(* Schneider Machine Expert - Basic project es5_6pompe_5max_6soglie_misura_livello_scelta_alternanza_spegnimento_graduale_o_livello_minimo, file version 3.0.0.0 *)
(* ProjectInformations: Name=New project *)

HARDWARE
  Cpu 0: TM221C40R
  ModuleExtensionObject 0: TM3AI8/G
  EthernetConfiguration: NetworkName=M221, IpAllocationMode=FixedAddress, IpAddress=0.0.0.0, SubnetMask=0.0.0.0
  SerialLineConfiguration: Baud=Baud19200, Parity=ParityEven, DataBits=DataBits8, StopBits=StopBits1, PhysicalMedium=PhysicalMediumRs485, TransmissionMode=TransmissionModeModbusRtu, SlaveId=1, Addressing=SlaveAddressing
  MastTask: UsePeriodScanMode=false, PeriodScan=100
  FastTask: Period=255
  CpuBehavior: StartingMode=StartAsPreviousState, AutoSaveRamOnEeprom=true, WatchdogPeriod=250

SYMBOLS  (address, symbol, comment, settings)
  %M0       P1_USABILE
  %M1       P2_USABILE
  %M2       P1_COMANDATA  "Stesso valore di P1_CMD. Permette di identificare gli edges, visto che P1_CMD non può farlo."
  %M3       P2_COMANDATA  "Stesso valore di P2_CMD. Permette di identificare gli edges, visto che P2_CMD non può farlo."
  %M4       P3_USABILE
  %M5       P4_USABILE
  %M6       P3_COMANDATA
  %M7       P4_COMANDATA
  %M8       ESISTE_PROX_POMPA_CON_MINOR_ORE  "Nel loop, può non esistere una prossima pompa usabile e non comandata con il minor numero ore."
  %M9       ORA_E_00  "E' mezzanotte?"
  %M10      DECISO_ORDINE  "In intervallo in cui alternare le pompe per altern. giorn., è stata deciso quale sarà prossima pompa con minor ore?"
  %M11      PRIMA_POMPA_COMANDATA  "La prima pompa dell'ordine è stata effettivamente comandata quando serviva?"
  %M12      SECONDA_POMPA_COMANDATA  "La seconda pompa dell'ordine è stata effettivamente comandata quando serviva?"
  %M13      TERZA_POMPA_COMANDATA  "La terza pompa dell'ordine è stata effettivamente comandata quando serviva?"
  %M14      SOTTO_SOGLIA_MIN1
  %M15      SOPRA_SOGLIA_MAX1
  %M16      SOPRA_SOGLIA_MAX2
  %M17      PASSATO_SOGLIA_MAX1
  %M18      PASSATO_SOGLIA_MAX2
  %M19      SOTTO_SOGLIA_MIN2
  %M20      PASSATO_SOGLIA_MAX3
  %M21      PASSATO_SOGLIA_MIN3
  %M22      SOTTO_SOGLIA_MIN3
  %M23      SOPRA_SOGLIA_MAX3
  %M24      P5_USABILE
  %M25        "(occupato, placeholder)"
  %M26      P6_USABILE
  %M27      P5_COMANDATA
  %M28      P6_COMANDATA
  %M29      QUARTA_POMPA_COMANDATA
  %M30      QUINTA_POMPA_COMANDATA
  %S6       SB_TB1S  "Time base of 1 s generated by an internal clock"
  %MW0      NUM_POMPE_DA_COMANDARE  "Numero di pompe da comandare in base alle soglie raggiunte."
  %MW1      NUM_POMPE_COMANDATE  "Numero di pompe effettivamente comandate, in base alle loro disponibilità."
  %MW2      NUM_POMPE  "Numero di pompe totali."
  %MW3      ULTIMO_MINOR_SECONDI_LAVORATI  "Ultimi secondi lavorati più piccoli (valore temporaneo, da usare solo nel loop)."
  %MW4      PROSSIMA_POMPA_DA_COMANDARE  "Numero da 1 a NUM_POMPE che indica la prossima pompa da comandare."
  %MW5      POMPA_ATTUALE_LOOP  "Pompa attuale nel loop."
  %MW6      NUM_POMPE_COMANDATE_MAX  "Num"
  %MW7      CONTA_POMPE_COMANDATE_MAX  "Da usare in loop e da resettare.  Assume il valore da 1 fino a NUM_POMPE_COMANDATE_MAX."
  %MW8      ORDINE_PRIMA_POMPA
  %MW9      ORDINE_SECONDA_POMPA
  %MW10     ORDINE_TERZA_POMPA
  %MW11     STRG_ALTERNANZA_ATTUALE
  %MW12     LVL_PERC
  %MW13     ORDINE_QUARTA_POMPA
  %MW14     ORDINE_QUINTA_POMPA
  %C0       CONTATORE_P1_SECONDI_LAVORATI  [Preset=0]
  %C1       CONTATORE_P2_SECONDI_LAVORATI  [Preset=0]
  %C2       CONTATORE_P3_SECONDI_LAVORATI  [Preset=0]
  %C3       CONTATORE_P4_SECONDI_LAVORATI  [Preset=0]
  %C4       CONTATORE_P5_SECONDI_LAVORATI  [Preset=0]
  %C5       CONTATORE_P6_SECONDI_LAVORATI  [Preset=0]
  %I0.0     P1_AUTO
  %I0.1     P1_MOTO
  %I0.2     P1_ANOMALIA
  %I0.3     P2_AUTO
  %I0.4     P2_MOTO
  %I0.5     P2_ANOMALIA
  %I0.9     P3_AUTO
  %I0.10    P3_MOTO
  %I0.11    P3_ANOMALIA
  %I0.12    P4_AUTO
  %I0.13    P4_MOTO
  %I0.14    P4_ANOMALIA
  %I0.15    P5_AUTO
  %I0.16    P5_MOTO
  %I0.17    P5_ANOMALIA
  %I0.18    P6_AUTO
  %I0.19    P6_MOTO
  %I0.20    P6_ANOMALIA
  %Q0.0     P1_CMD
  %Q0.1     P2_CMD
  %Q0.2     P3_CMD
  %Q0.3     P4_CMD
  %Q0.4     ERR_STRG_ALTERNANZA_INVALIDA
  %Q0.5     P5_CMD
  %Q0.6     P6_CMD
  %IW0.0    IO_STRG_ALTERNANZA  "0 = livello minimo; 1 = spegnimento graduale;"  [Type=Type_0_10V, Scope=Scope_Normal, Minimum=0, Maximum=1000]
  %IW1.0    IO_LVL  [Type=Type_4_20mA, Scope=Scope_Customized, Minimum=4000, Maximum=20000]
  %IW1.1    SOGLIA_MIN1_PERC  [Type=Type_0_10V, Scope=Scope_Customized, Minimum=0, Maximum=100]
  %IW1.2    SOGLIA_MAX1_PERC  [Type=Type_0_10V, Scope=Scope_Customized, Minimum=0, Maximum=100]
  %IW1.3    SOGLIA_MIN2_PERC  [Type=Type_0_10V, Scope=Scope_Customized, Minimum=0, Maximum=100]
  %IW1.4    SOGLIA_MAX2_PERC  [Type=Type_0_10V, Scope=Scope_Customized, Minimum=0, Maximum=100]
  %IW1.5    SOGLIA_MIN3_PERC  [Type=Type_0_10V, Scope=Scope_Customized, Minimum=0, Maximum=100]
  %IW1.6    SOGLIA_MAX3_PERC  [Type=Type_0_10V, Scope=Scope_Customized, Minimum=0, Maximum=100]

POU Main
  (* SectionNumber=1 *)

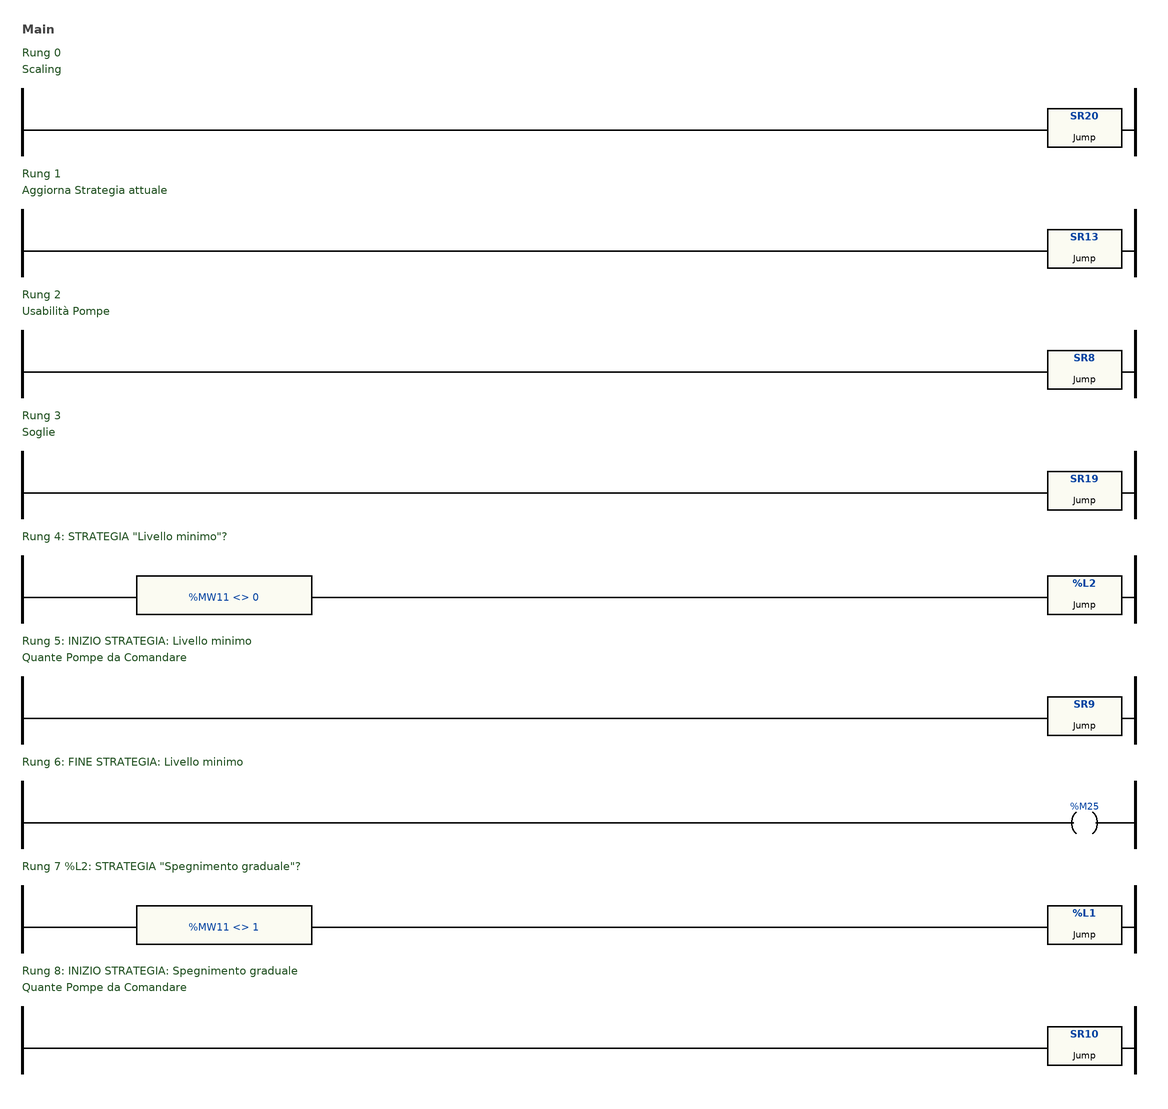

// Rung 0
// Scaling
  LD 1
  SR20
  // as ST:
  //   SR20();

// Rung 1
// Aggiorna Strategia attuale
  LD 1
  SR13
  // as ST:
  //   SR13();

// Rung 2
// Usabilità Pompe
  LD 1
  SR8
  // as ST:
  //   SR8();

// Rung 3
// Soglie
  LD 1
  SR19
  // as ST:
  //   SR19();

// Rung 4: STRATEGIA "Livello minimo"?
  LD [ %MW11 <> 0 ]       (* STRG_ALTERNANZA_ATTUALE *)
  JMPC %L2
  // as ST:
  //   IF STRG_ALTERNANZA_ATTUALE <> 0 THEN JMP %L2; END_IF;

// Rung 5: INIZIO STRATEGIA: Livello minimo
// Quante Pompe da Comandare
  LD 1
  SR9
  // as ST:
  //   SR9();

// Rung 6: FINE STRATEGIA: Livello minimo
  LD 1
  ST %M25
  // as ST:
  //   %M25 := TRUE;

// Rung 7 %L2: STRATEGIA "Spegnimento graduale"?
  %L2:
  LD [ %MW11 <> 1 ]       (* STRG_ALTERNANZA_ATTUALE *)
  JMPC %L1
  // as ST:
  //   %L2:
  //   IF STRG_ALTERNANZA_ATTUALE <> 1 THEN JMP %L1; END_IF;

// Rung 8: INIZIO STRATEGIA: Spegnimento graduale
// Quante Pompe da Comandare
  LD 1
  SR10
  // as ST:
  //   SR10();

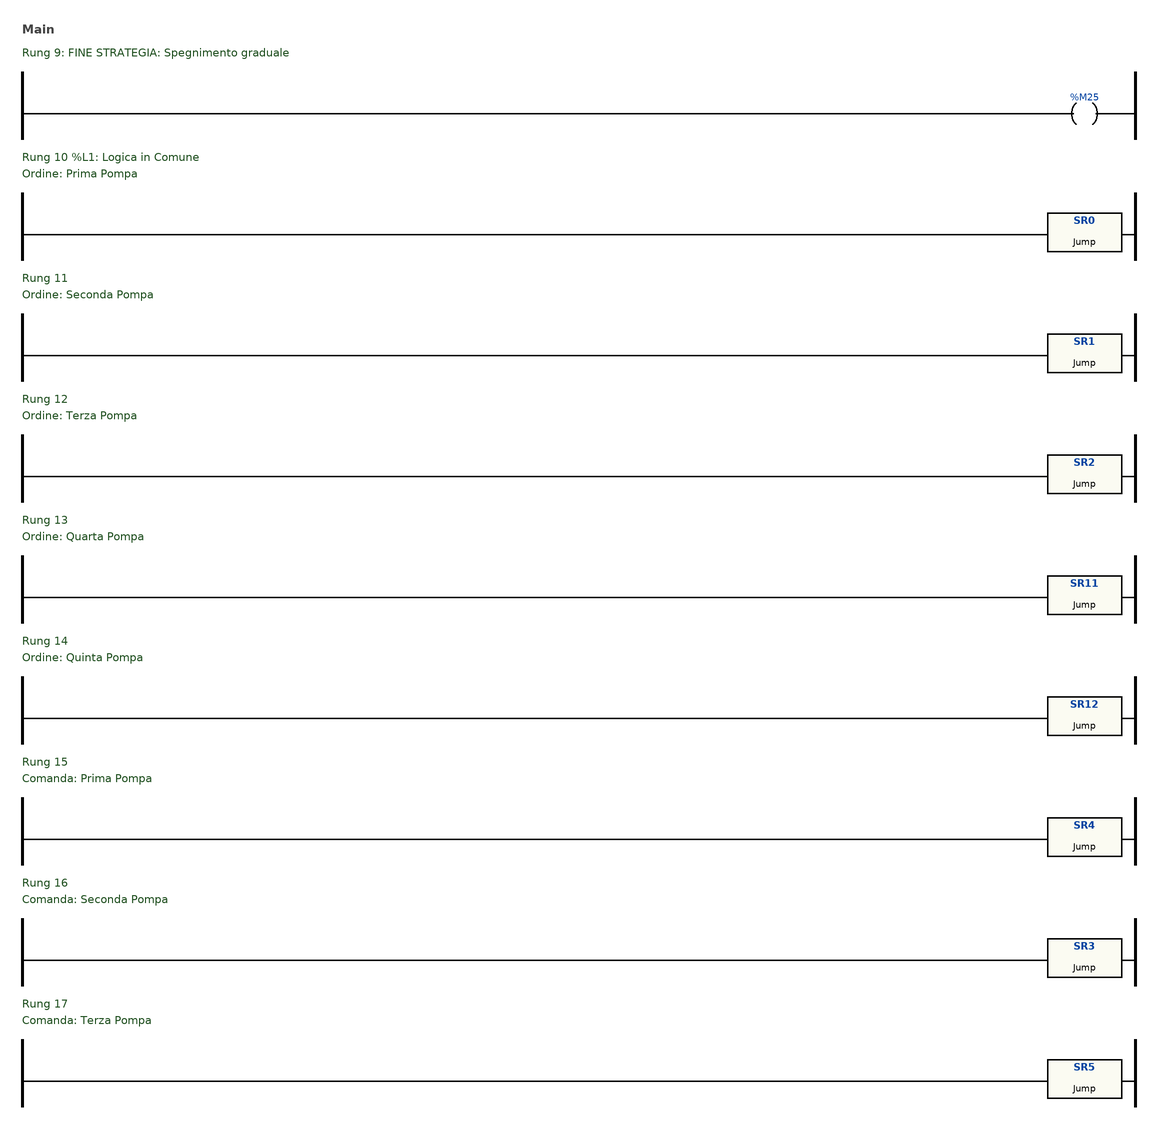

// Rung 9: FINE STRATEGIA: Spegnimento graduale
  LD 1
  ST %M25
  // as ST:
  //   %M25 := TRUE;

// Rung 10 %L1: Logica in Comune
// Ordine: Prima Pompa
  %L1:
  LD 1
  SR0
  // as ST:
  //   %L1:
  //   SR0();

// Rung 11
// Ordine: Seconda Pompa
  LD 1
  SR1
  // as ST:
  //   SR1();

// Rung 12
// Ordine: Terza Pompa
  LD 1
  SR2
  // as ST:
  //   SR2();

// Rung 13
// Ordine: Quarta Pompa
  LD 1
  SR11
  // as ST:
  //   SR11();

// Rung 14
// Ordine: Quinta Pompa
  LD 1
  SR12
  // as ST:
  //   SR12();

// Rung 15
// Comanda: Prima Pompa
  LD 1
  SR4
  // as ST:
  //   SR4();

// Rung 16
// Comanda: Seconda Pompa
  LD 1
  SR3
  // as ST:
  //   SR3();

// Rung 17
// Comanda: Terza Pompa
  LD 1
  SR5
  // as ST:
  //   SR5();

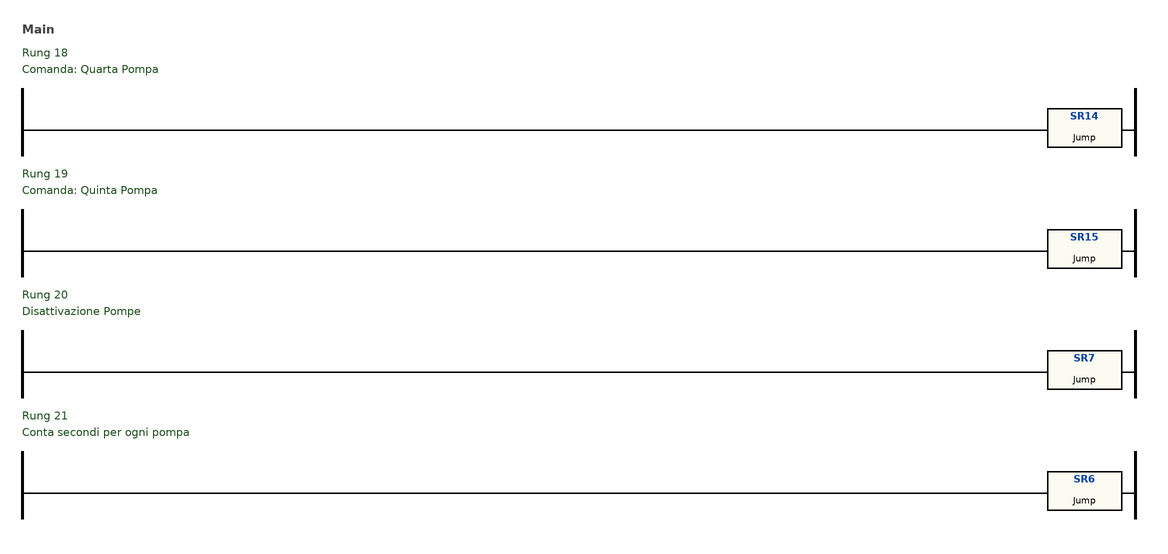

// Rung 18
// Comanda: Quarta Pompa
  LD 1
  SR14
  // as ST:
  //   SR14();

// Rung 19
// Comanda: Quinta Pompa
  LD 1
  SR15
  // as ST:
  //   SR15();

// Rung 20
// Disattivazione Pompe
  LD 1
  SR7
  // as ST:
  //   SR7();

// Rung 21
// Conta secondi per ogni pompa
  LD 1
  SR6
  // as ST:
  //   SR6();

Subroutine Ordine: Prima Pompa
  (* SectionNumber=2, Number=0 *)

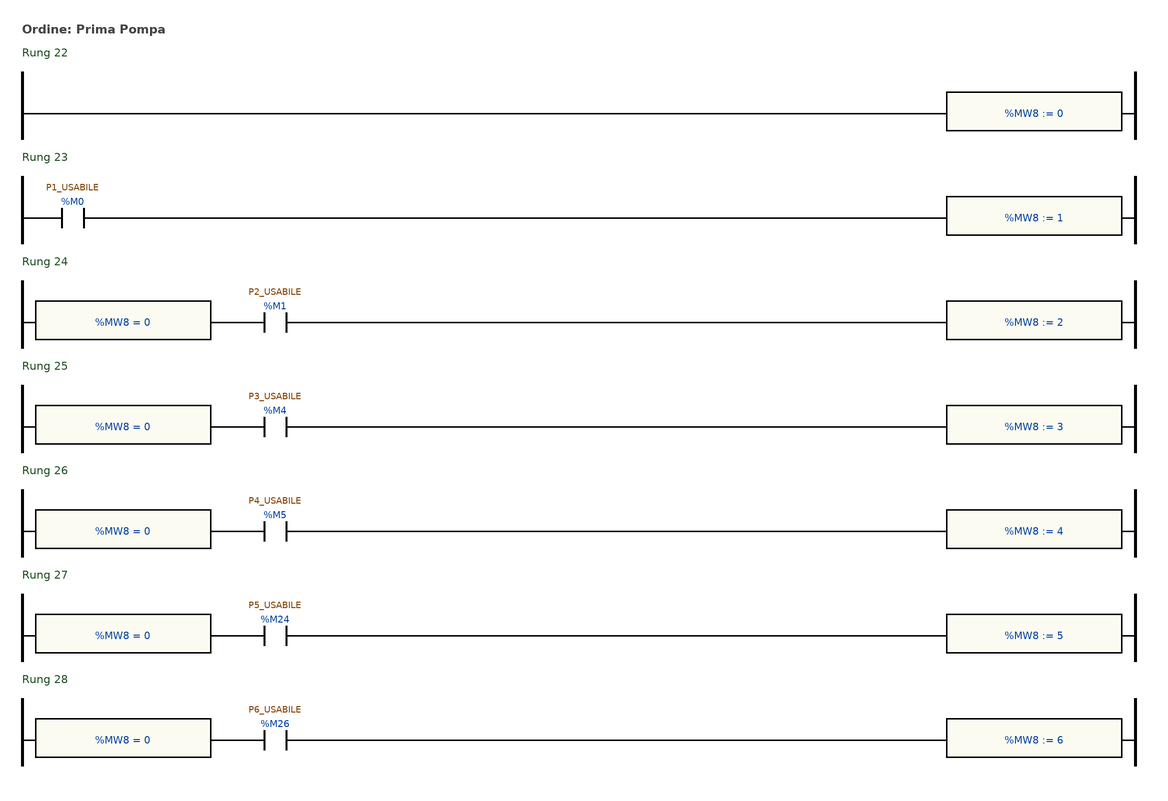

// Rung 22
  LD 1
  [ %MW8 := 0 ]           (* ORDINE_PRIMA_POMPA *)
  // as ST:
  //   ORDINE_PRIMA_POMPA := 0;

// Rung 23
  LD %M0                  (* P1_USABILE *)
  [ %MW8 := 1 ]           (* ORDINE_PRIMA_POMPA *)
  // as ST:
  //   IF P1_USABILE THEN ORDINE_PRIMA_POMPA := 1; END_IF;

// Rung 24
  LD [ %MW8 = 0 ]         (* ORDINE_PRIMA_POMPA *)
  AND %M1                 (* P2_USABILE *)
  [ %MW8 := 2 ]           (* ORDINE_PRIMA_POMPA *)
  // as ST:
  //   IF ORDINE_PRIMA_POMPA = 0 AND P2_USABILE THEN ORDINE_PRIMA_POMPA := 2; END_IF;

// Rung 25
  LD [ %MW8 = 0 ]         (* ORDINE_PRIMA_POMPA *)
  AND %M4                 (* P3_USABILE *)
  [ %MW8 := 3 ]           (* ORDINE_PRIMA_POMPA *)
  // as ST:
  //   IF ORDINE_PRIMA_POMPA = 0 AND P3_USABILE THEN ORDINE_PRIMA_POMPA := 3; END_IF;

// Rung 26
  LD [ %MW8 = 0 ]         (* ORDINE_PRIMA_POMPA *)
  AND %M5                 (* P4_USABILE *)
  [ %MW8 := 4 ]           (* ORDINE_PRIMA_POMPA *)
  // as ST:
  //   IF ORDINE_PRIMA_POMPA = 0 AND P4_USABILE THEN ORDINE_PRIMA_POMPA := 4; END_IF;

// Rung 27
  LD [ %MW8 = 0 ]         (* ORDINE_PRIMA_POMPA *)
  AND %M24                (* P5_USABILE *)
  [ %MW8 := 5 ]           (* ORDINE_PRIMA_POMPA *)
  // as ST:
  //   IF ORDINE_PRIMA_POMPA = 0 AND P5_USABILE THEN ORDINE_PRIMA_POMPA := 5; END_IF;

// Rung 28
  LD [ %MW8 = 0 ]         (* ORDINE_PRIMA_POMPA *)
  AND %M26                (* P6_USABILE *)
  [ %MW8 := 6 ]           (* ORDINE_PRIMA_POMPA *)
  // as ST:
  //   IF ORDINE_PRIMA_POMPA = 0 AND P6_USABILE THEN ORDINE_PRIMA_POMPA := 6; END_IF;

Subroutine Ordine: Seconda Pompa
  (* SectionNumber=3, Number=1 *)

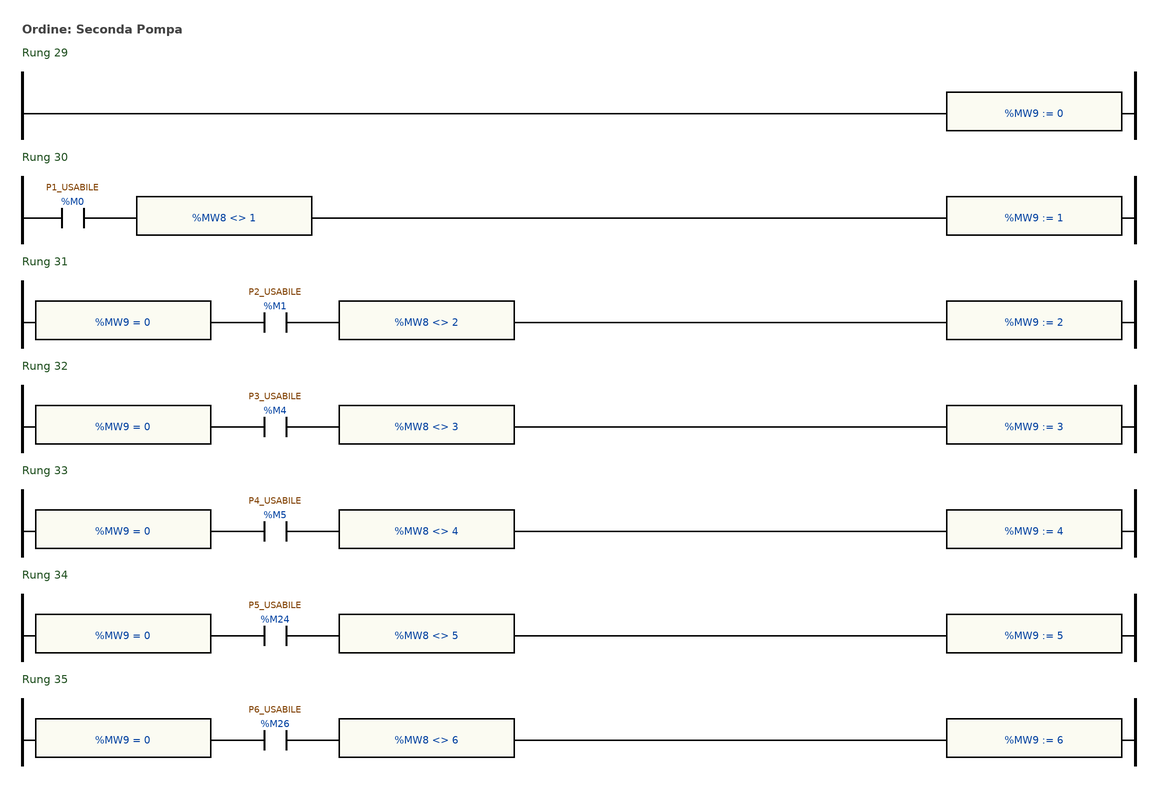

// Rung 29
  LD 1
  [ %MW9 := 0 ]           (* ORDINE_SECONDA_POMPA *)
  // as ST:
  //   ORDINE_SECONDA_POMPA := 0;

// Rung 30
  LD %M0                  (* P1_USABILE *)
  AND [ %MW8 <> 1 ]       (* ORDINE_PRIMA_POMPA *)
  [ %MW9 := 1 ]           (* ORDINE_SECONDA_POMPA *)
  // as ST:
  //   IF P1_USABILE AND ORDINE_PRIMA_POMPA <> 1 THEN ORDINE_SECONDA_POMPA := 1; END_IF;

// Rung 31
  LD [ %MW9 = 0 ]         (* ORDINE_SECONDA_POMPA *)
  AND %M1                 (* P2_USABILE *)
  AND [ %MW8 <> 2 ]       (* ORDINE_PRIMA_POMPA *)
  [ %MW9 := 2 ]           (* ORDINE_SECONDA_POMPA *)
  // as ST:
  //   IF ORDINE_SECONDA_POMPA = 0 AND P2_USABILE AND ORDINE_PRIMA_POMPA <> 2 THEN ORDINE_SECONDA_POMPA := 2; END_IF;

// Rung 32
  LD [ %MW9 = 0 ]         (* ORDINE_SECONDA_POMPA *)
  AND %M4                 (* P3_USABILE *)
  AND [ %MW8 <> 3 ]       (* ORDINE_PRIMA_POMPA *)
  [ %MW9 := 3 ]           (* ORDINE_SECONDA_POMPA *)
  // as ST:
  //   IF ORDINE_SECONDA_POMPA = 0 AND P3_USABILE AND ORDINE_PRIMA_POMPA <> 3 THEN ORDINE_SECONDA_POMPA := 3; END_IF;

// Rung 33
  LD [ %MW9 = 0 ]         (* ORDINE_SECONDA_POMPA *)
  AND %M5                 (* P4_USABILE *)
  AND [ %MW8 <> 4 ]       (* ORDINE_PRIMA_POMPA *)
  [ %MW9 := 4 ]           (* ORDINE_SECONDA_POMPA *)
  // as ST:
  //   IF ORDINE_SECONDA_POMPA = 0 AND P4_USABILE AND ORDINE_PRIMA_POMPA <> 4 THEN ORDINE_SECONDA_POMPA := 4; END_IF;

// Rung 34
  LD [ %MW9 = 0 ]         (* ORDINE_SECONDA_POMPA *)
  AND %M24                (* P5_USABILE *)
  AND [ %MW8 <> 5 ]       (* ORDINE_PRIMA_POMPA *)
  [ %MW9 := 5 ]           (* ORDINE_SECONDA_POMPA *)
  // as ST:
  //   IF ORDINE_SECONDA_POMPA = 0 AND P5_USABILE AND ORDINE_PRIMA_POMPA <> 5 THEN ORDINE_SECONDA_POMPA := 5; END_IF;

// Rung 35
  LD [ %MW9 = 0 ]         (* ORDINE_SECONDA_POMPA *)
  AND %M26                (* P6_USABILE *)
  AND [ %MW8 <> 6 ]       (* ORDINE_PRIMA_POMPA *)
  [ %MW9 := 6 ]           (* ORDINE_SECONDA_POMPA *)
  // as ST:
  //   IF ORDINE_SECONDA_POMPA = 0 AND P6_USABILE AND ORDINE_PRIMA_POMPA <> 6 THEN ORDINE_SECONDA_POMPA := 6; END_IF;

Subroutine Ordine: Terza Pompa
  (* SectionNumber=4, Number=2 *)

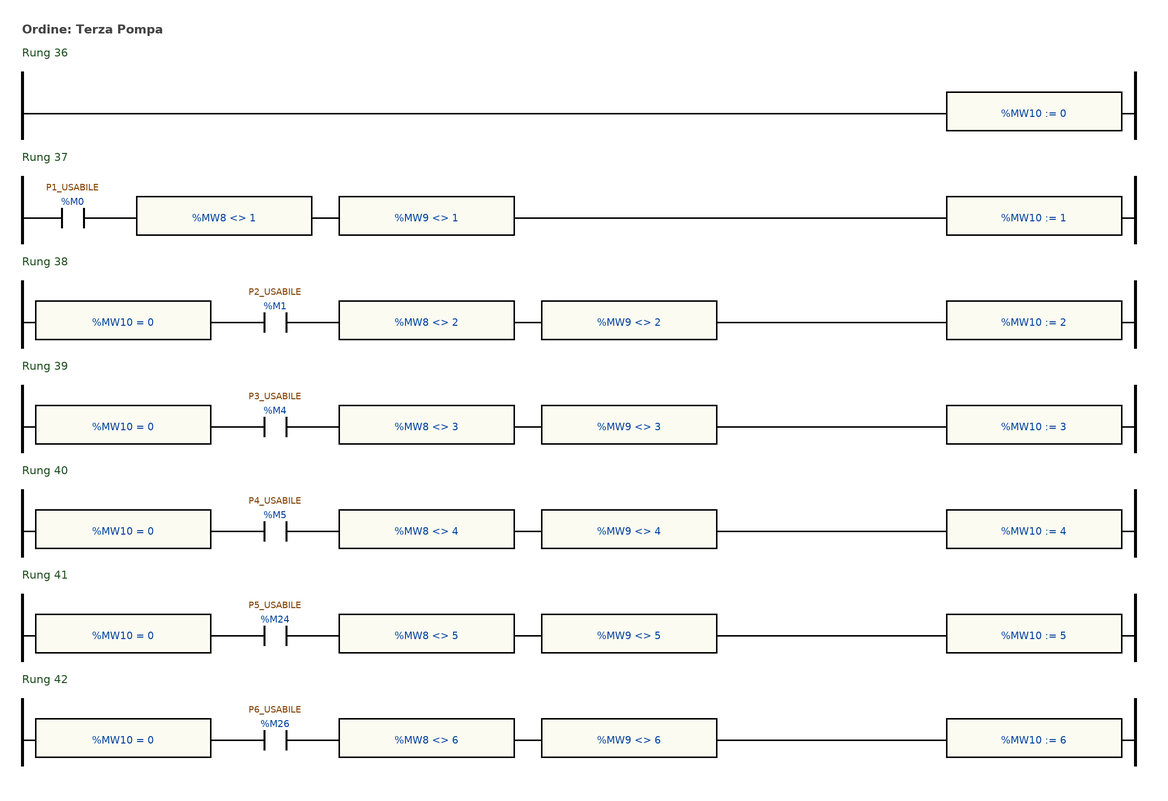

// Rung 36
  LD 1
  [ %MW10 := 0 ]          (* ORDINE_TERZA_POMPA *)
  // as ST:
  //   ORDINE_TERZA_POMPA := 0;

// Rung 37
  LD %M0                  (* P1_USABILE *)
  AND [ %MW8 <> 1 ]       (* ORDINE_PRIMA_POMPA *)
  AND [ %MW9 <> 1 ]       (* ORDINE_SECONDA_POMPA *)
  [ %MW10 := 1 ]          (* ORDINE_TERZA_POMPA *)
  // as ST:
  //   IF P1_USABILE AND ORDINE_PRIMA_POMPA <> 1 AND ORDINE_SECONDA_POMPA <> 1 THEN ORDINE_TERZA_POMPA := 1; END_IF;

// Rung 38
  LD [ %MW10 = 0 ]        (* ORDINE_TERZA_POMPA *)
  AND %M1                 (* P2_USABILE *)
  AND [ %MW8 <> 2 ]       (* ORDINE_PRIMA_POMPA *)
  AND [ %MW9 <> 2 ]       (* ORDINE_SECONDA_POMPA *)
  [ %MW10 := 2 ]          (* ORDINE_TERZA_POMPA *)
  // as ST:
  //   IF ORDINE_TERZA_POMPA = 0 AND P2_USABILE AND ORDINE_PRIMA_POMPA <> 2 AND ORDINE_SECONDA_POMPA <> 2 THEN ORDINE_TERZA_POMPA := 2; END_IF;

// Rung 39
  LD [ %MW10 = 0 ]        (* ORDINE_TERZA_POMPA *)
  AND %M4                 (* P3_USABILE *)
  AND [ %MW8 <> 3 ]       (* ORDINE_PRIMA_POMPA *)
  AND [ %MW9 <> 3 ]       (* ORDINE_SECONDA_POMPA *)
  [ %MW10 := 3 ]          (* ORDINE_TERZA_POMPA *)
  // as ST:
  //   IF ORDINE_TERZA_POMPA = 0 AND P3_USABILE AND ORDINE_PRIMA_POMPA <> 3 AND ORDINE_SECONDA_POMPA <> 3 THEN ORDINE_TERZA_POMPA := 3; END_IF;

// Rung 40
  LD [ %MW10 = 0 ]        (* ORDINE_TERZA_POMPA *)
  AND %M5                 (* P4_USABILE *)
  AND [ %MW8 <> 4 ]       (* ORDINE_PRIMA_POMPA *)
  AND [ %MW9 <> 4 ]       (* ORDINE_SECONDA_POMPA *)
  [ %MW10 := 4 ]          (* ORDINE_TERZA_POMPA *)
  // as ST:
  //   IF ORDINE_TERZA_POMPA = 0 AND P4_USABILE AND ORDINE_PRIMA_POMPA <> 4 AND ORDINE_SECONDA_POMPA <> 4 THEN ORDINE_TERZA_POMPA := 4; END_IF;

// Rung 41
  LD [ %MW10 = 0 ]        (* ORDINE_TERZA_POMPA *)
  AND %M24                (* P5_USABILE *)
  AND [ %MW8 <> 5 ]       (* ORDINE_PRIMA_POMPA *)
  AND [ %MW9 <> 5 ]       (* ORDINE_SECONDA_POMPA *)
  [ %MW10 := 5 ]          (* ORDINE_TERZA_POMPA *)
  // as ST:
  //   IF ORDINE_TERZA_POMPA = 0 AND P5_USABILE AND ORDINE_PRIMA_POMPA <> 5 AND ORDINE_SECONDA_POMPA <> 5 THEN ORDINE_TERZA_POMPA := 5; END_IF;

// Rung 42
  LD [ %MW10 = 0 ]        (* ORDINE_TERZA_POMPA *)
  AND %M26                (* P6_USABILE *)
  AND [ %MW8 <> 6 ]       (* ORDINE_PRIMA_POMPA *)
  AND [ %MW9 <> 6 ]       (* ORDINE_SECONDA_POMPA *)
  [ %MW10 := 6 ]          (* ORDINE_TERZA_POMPA *)
  // as ST:
  //   IF ORDINE_TERZA_POMPA = 0 AND P6_USABILE AND ORDINE_PRIMA_POMPA <> 6 AND ORDINE_SECONDA_POMPA <> 6 THEN ORDINE_TERZA_POMPA := 6; END_IF;

Subroutine Comanda: Prima Pompa
  (* SectionNumber=5, Number=4 *)

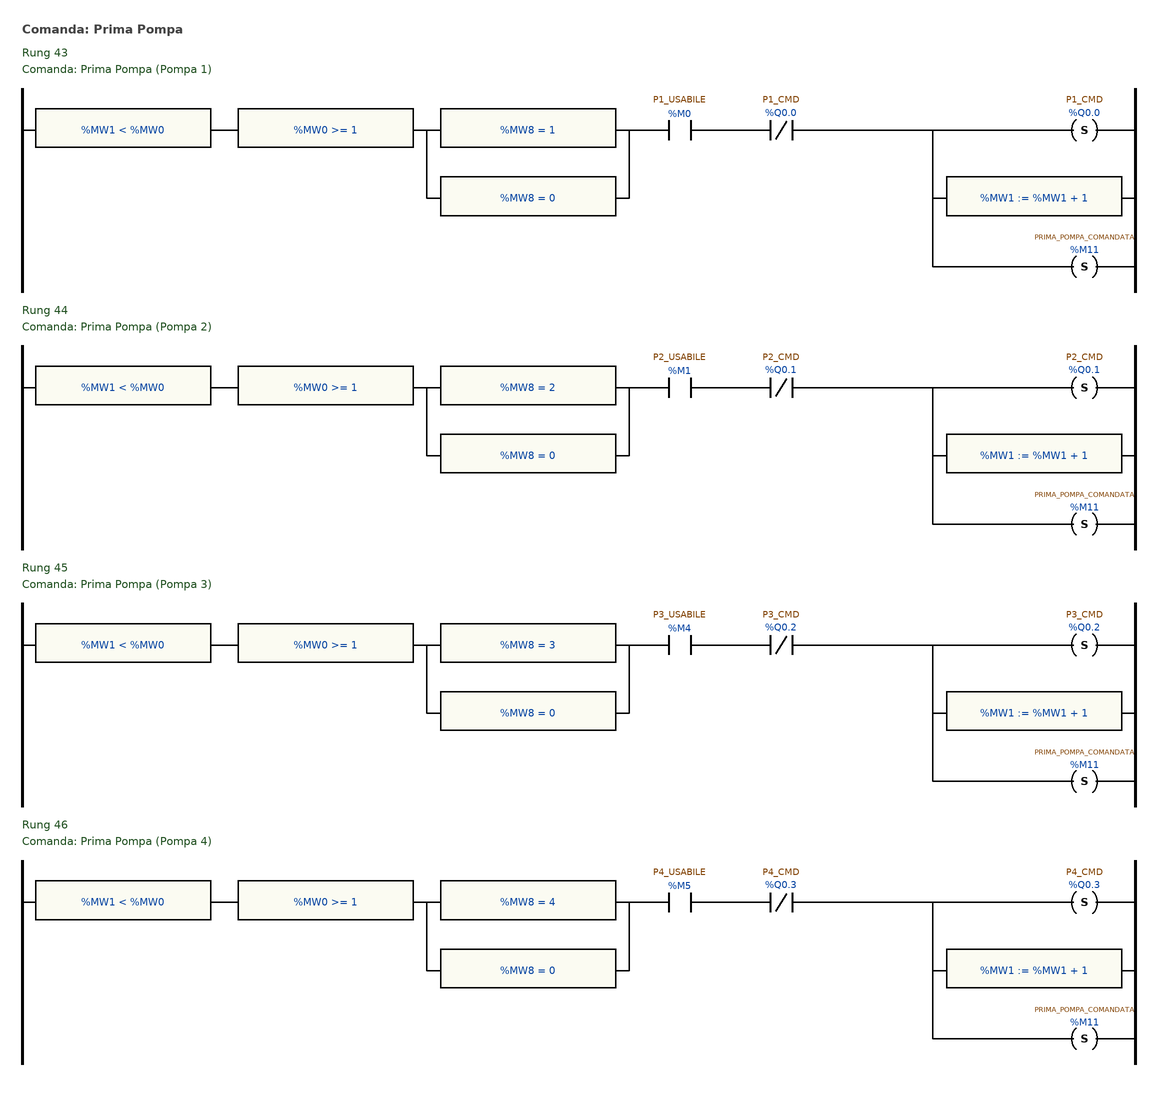

// Rung 43
// Comanda: Prima Pompa (Pompa 1)
  LD [ %MW1 < %MW0 ]      (* NUM_POMPE_COMANDATE, NUM_POMPE_DA_COMANDARE *)
  AND [ %MW0 >= 1 ]       (* NUM_POMPE_DA_COMANDARE *)
  AND( [ %MW8 = 1 ]       (* ORDINE_PRIMA_POMPA *)
  OR [ %MW8 = 0 ]         (* ORDINE_PRIMA_POMPA *)
  )
  AND %M0                 (* P1_USABILE *)
  ANDN %Q0.0              (* P1_CMD *)
  S %Q0.0                 (* P1_CMD *)
  [ %MW1 := %MW1 + 1 ]    (* NUM_POMPE_COMANDATE, NUM_POMPE_COMANDATE *)
  S %M11                  (* PRIMA_POMPA_COMANDATA *)
  // as ST:
  //   _t1 := NUM_POMPE_COMANDATE < NUM_POMPE_DA_COMANDARE AND NUM_POMPE_DA_COMANDARE >= 1 AND (ORDINE_PRIMA_POMPA = 1 OR ORDINE_PRIMA_POMPA = 0) AND P1_USABILE AND NOT P1_CMD;
  //   IF _t1 THEN P1_CMD := TRUE; END_IF;
  //   IF _t1 THEN NUM_POMPE_COMANDATE := NUM_POMPE_COMANDATE + 1; END_IF;
  //   IF _t1 THEN PRIMA_POMPA_COMANDATA := TRUE; END_IF;

// Rung 44
// Comanda: Prima Pompa (Pompa 2)
  LD [ %MW1 < %MW0 ]      (* NUM_POMPE_COMANDATE, NUM_POMPE_DA_COMANDARE *)
  AND [ %MW0 >= 1 ]       (* NUM_POMPE_DA_COMANDARE *)
  AND( [ %MW8 = 2 ]       (* ORDINE_PRIMA_POMPA *)
  OR [ %MW8 = 0 ]         (* ORDINE_PRIMA_POMPA *)
  )
  AND %M1                 (* P2_USABILE *)
  ANDN %Q0.1              (* P2_CMD *)
  S %Q0.1                 (* P2_CMD *)
  [ %MW1 := %MW1 + 1 ]    (* NUM_POMPE_COMANDATE, NUM_POMPE_COMANDATE *)
  S %M11                  (* PRIMA_POMPA_COMANDATA *)
  // as ST:
  //   _t1 := NUM_POMPE_COMANDATE < NUM_POMPE_DA_COMANDARE AND NUM_POMPE_DA_COMANDARE >= 1 AND (ORDINE_PRIMA_POMPA = 2 OR ORDINE_PRIMA_POMPA = 0) AND P2_USABILE AND NOT P2_CMD;
  //   IF _t1 THEN P2_CMD := TRUE; END_IF;
  //   IF _t1 THEN NUM_POMPE_COMANDATE := NUM_POMPE_COMANDATE + 1; END_IF;
  //   IF _t1 THEN PRIMA_POMPA_COMANDATA := TRUE; END_IF;

// Rung 45
// Comanda: Prima Pompa (Pompa 3)
  LD [ %MW1 < %MW0 ]      (* NUM_POMPE_COMANDATE, NUM_POMPE_DA_COMANDARE *)
  AND [ %MW0 >= 1 ]       (* NUM_POMPE_DA_COMANDARE *)
  AND( [ %MW8 = 3 ]       (* ORDINE_PRIMA_POMPA *)
  OR [ %MW8 = 0 ]         (* ORDINE_PRIMA_POMPA *)
  )
  AND %M4                 (* P3_USABILE *)
  ANDN %Q0.2              (* P3_CMD *)
  S %Q0.2                 (* P3_CMD *)
  [ %MW1 := %MW1 + 1 ]    (* NUM_POMPE_COMANDATE, NUM_POMPE_COMANDATE *)
  S %M11                  (* PRIMA_POMPA_COMANDATA *)
  // as ST:
  //   _t1 := NUM_POMPE_COMANDATE < NUM_POMPE_DA_COMANDARE AND NUM_POMPE_DA_COMANDARE >= 1 AND (ORDINE_PRIMA_POMPA = 3 OR ORDINE_PRIMA_POMPA = 0) AND P3_USABILE AND NOT P3_CMD;
  //   IF _t1 THEN P3_CMD := TRUE; END_IF;
  //   IF _t1 THEN NUM_POMPE_COMANDATE := NUM_POMPE_COMANDATE + 1; END_IF;
  //   IF _t1 THEN PRIMA_POMPA_COMANDATA := TRUE; END_IF;

// Rung 46
// Comanda: Prima Pompa (Pompa 4)
  LD [ %MW1 < %MW0 ]      (* NUM_POMPE_COMANDATE, NUM_POMPE_DA_COMANDARE *)
  AND [ %MW0 >= 1 ]       (* NUM_POMPE_DA_COMANDARE *)
  AND( [ %MW8 = 4 ]       (* ORDINE_PRIMA_POMPA *)
  OR [ %MW8 = 0 ]         (* ORDINE_PRIMA_POMPA *)
  )
  AND %M5                 (* P4_USABILE *)
  ANDN %Q0.3              (* P4_CMD *)
  S %Q0.3                 (* P4_CMD *)
  [ %MW1 := %MW1 + 1 ]    (* NUM_POMPE_COMANDATE, NUM_POMPE_COMANDATE *)
  S %M11                  (* PRIMA_POMPA_COMANDATA *)
  // as ST:
  //   _t1 := NUM_POMPE_COMANDATE < NUM_POMPE_DA_COMANDARE AND NUM_POMPE_DA_COMANDARE >= 1 AND (ORDINE_PRIMA_POMPA = 4 OR ORDINE_PRIMA_POMPA = 0) AND P4_USABILE AND NOT P4_CMD;
  //   IF _t1 THEN P4_CMD := TRUE; END_IF;
  //   IF _t1 THEN NUM_POMPE_COMANDATE := NUM_POMPE_COMANDATE + 1; END_IF;
  //   IF _t1 THEN PRIMA_POMPA_COMANDATA := TRUE; END_IF;

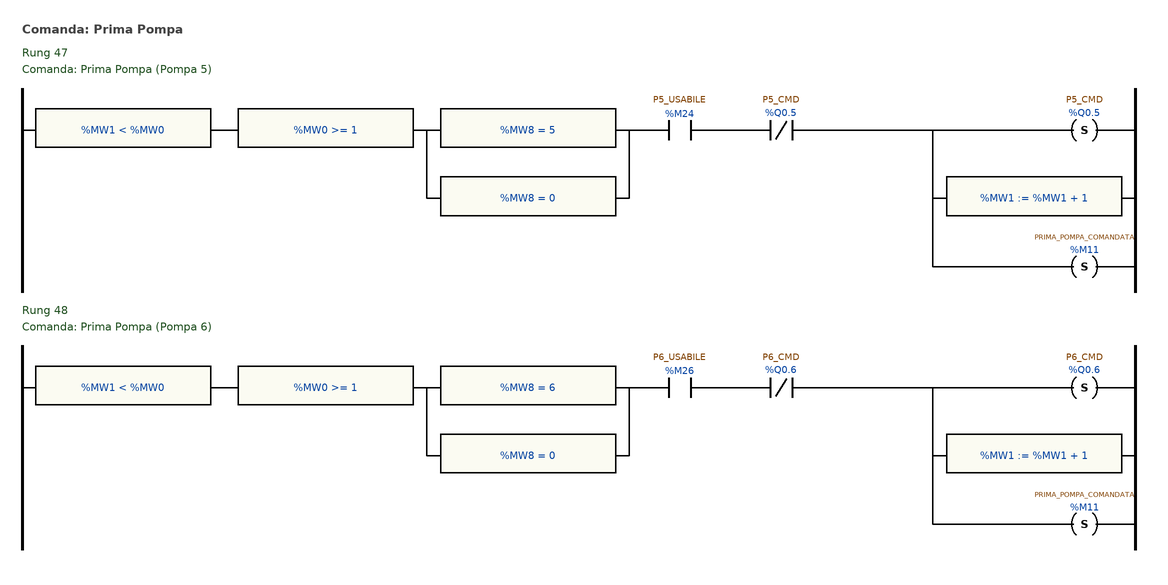

// Rung 47
// Comanda: Prima Pompa (Pompa 5)
  LD [ %MW1 < %MW0 ]      (* NUM_POMPE_COMANDATE, NUM_POMPE_DA_COMANDARE *)
  AND [ %MW0 >= 1 ]       (* NUM_POMPE_DA_COMANDARE *)
  AND( [ %MW8 = 5 ]       (* ORDINE_PRIMA_POMPA *)
  OR [ %MW8 = 0 ]         (* ORDINE_PRIMA_POMPA *)
  )
  AND %M24                (* P5_USABILE *)
  ANDN %Q0.5              (* P5_CMD *)
  S %Q0.5                 (* P5_CMD *)
  [ %MW1 := %MW1 + 1 ]    (* NUM_POMPE_COMANDATE, NUM_POMPE_COMANDATE *)
  S %M11                  (* PRIMA_POMPA_COMANDATA *)
  // as ST:
  //   _t1 := NUM_POMPE_COMANDATE < NUM_POMPE_DA_COMANDARE AND NUM_POMPE_DA_COMANDARE >= 1 AND (ORDINE_PRIMA_POMPA = 5 OR ORDINE_PRIMA_POMPA = 0) AND P5_USABILE AND NOT P5_CMD;
  //   IF _t1 THEN P5_CMD := TRUE; END_IF;
  //   IF _t1 THEN NUM_POMPE_COMANDATE := NUM_POMPE_COMANDATE + 1; END_IF;
  //   IF _t1 THEN PRIMA_POMPA_COMANDATA := TRUE; END_IF;

// Rung 48
// Comanda: Prima Pompa (Pompa 6)
  LD [ %MW1 < %MW0 ]      (* NUM_POMPE_COMANDATE, NUM_POMPE_DA_COMANDARE *)
  AND [ %MW0 >= 1 ]       (* NUM_POMPE_DA_COMANDARE *)
  AND( [ %MW8 = 6 ]       (* ORDINE_PRIMA_POMPA *)
  OR [ %MW8 = 0 ]         (* ORDINE_PRIMA_POMPA *)
  )
  AND %M26                (* P6_USABILE *)
  ANDN %Q0.6              (* P6_CMD *)
  S %Q0.6                 (* P6_CMD *)
  [ %MW1 := %MW1 + 1 ]    (* NUM_POMPE_COMANDATE, NUM_POMPE_COMANDATE *)
  S %M11                  (* PRIMA_POMPA_COMANDATA *)
  // as ST:
  //   _t1 := NUM_POMPE_COMANDATE < NUM_POMPE_DA_COMANDARE AND NUM_POMPE_DA_COMANDARE >= 1 AND (ORDINE_PRIMA_POMPA = 6 OR ORDINE_PRIMA_POMPA = 0) AND P6_USABILE AND NOT P6_CMD;
  //   IF _t1 THEN P6_CMD := TRUE; END_IF;
  //   IF _t1 THEN NUM_POMPE_COMANDATE := NUM_POMPE_COMANDATE + 1; END_IF;
  //   IF _t1 THEN PRIMA_POMPA_COMANDATA := TRUE; END_IF;

Subroutine Comanda: Seconda Pompa
  (* SectionNumber=6, Number=3 *)

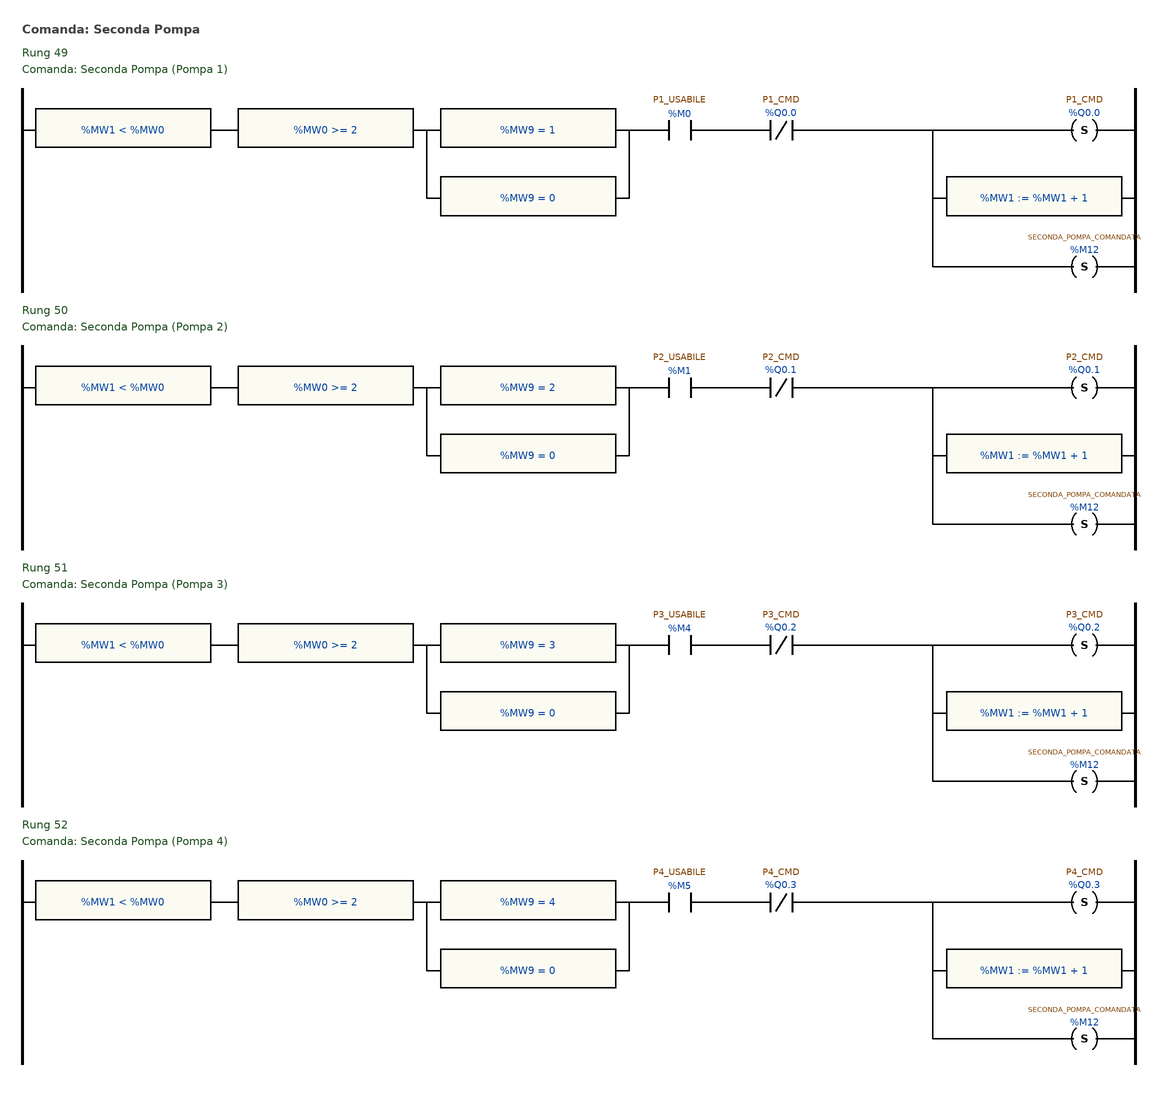

// Rung 49
// Comanda: Seconda Pompa (Pompa 1)
  LD [ %MW1 < %MW0 ]      (* NUM_POMPE_COMANDATE, NUM_POMPE_DA_COMANDARE *)
  AND [ %MW0 >= 2 ]       (* NUM_POMPE_DA_COMANDARE *)
  AND( [ %MW9 = 1 ]       (* ORDINE_SECONDA_POMPA *)
  OR [ %MW9 = 0 ]         (* ORDINE_SECONDA_POMPA *)
  )
  AND %M0                 (* P1_USABILE *)
  ANDN %Q0.0              (* P1_CMD *)
  S %Q0.0                 (* P1_CMD *)
  [ %MW1 := %MW1 + 1 ]    (* NUM_POMPE_COMANDATE, NUM_POMPE_COMANDATE *)
  S %M12                  (* SECONDA_POMPA_COMANDATA *)
  // as ST:
  //   _t1 := NUM_POMPE_COMANDATE < NUM_POMPE_DA_COMANDARE AND NUM_POMPE_DA_COMANDARE >= 2 AND (ORDINE_SECONDA_POMPA = 1 OR ORDINE_SECONDA_POMPA = 0) AND P1_USABILE AND NOT P1_CMD;
  //   IF _t1 THEN P1_CMD := TRUE; END_IF;
  //   IF _t1 THEN NUM_POMPE_COMANDATE := NUM_POMPE_COMANDATE + 1; END_IF;
  //   IF _t1 THEN SECONDA_POMPA_COMANDATA := TRUE; END_IF;

// Rung 50
// Comanda: Seconda Pompa (Pompa 2)
  LD [ %MW1 < %MW0 ]      (* NUM_POMPE_COMANDATE, NUM_POMPE_DA_COMANDARE *)
  AND [ %MW0 >= 2 ]       (* NUM_POMPE_DA_COMANDARE *)
  AND( [ %MW9 = 2 ]       (* ORDINE_SECONDA_POMPA *)
  OR [ %MW9 = 0 ]         (* ORDINE_SECONDA_POMPA *)
  )
  AND %M1                 (* P2_USABILE *)
  ANDN %Q0.1              (* P2_CMD *)
  S %Q0.1                 (* P2_CMD *)
  [ %MW1 := %MW1 + 1 ]    (* NUM_POMPE_COMANDATE, NUM_POMPE_COMANDATE *)
  S %M12                  (* SECONDA_POMPA_COMANDATA *)
  // as ST:
  //   _t1 := NUM_POMPE_COMANDATE < NUM_POMPE_DA_COMANDARE AND NUM_POMPE_DA_COMANDARE >= 2 AND (ORDINE_SECONDA_POMPA = 2 OR ORDINE_SECONDA_POMPA = 0) AND P2_USABILE AND NOT P2_CMD;
  //   IF _t1 THEN P2_CMD := TRUE; END_IF;
  //   IF _t1 THEN NUM_POMPE_COMANDATE := NUM_POMPE_COMANDATE + 1; END_IF;
  //   IF _t1 THEN SECONDA_POMPA_COMANDATA := TRUE; END_IF;

// Rung 51
// Comanda: Seconda Pompa (Pompa 3)
  LD [ %MW1 < %MW0 ]      (* NUM_POMPE_COMANDATE, NUM_POMPE_DA_COMANDARE *)
  AND [ %MW0 >= 2 ]       (* NUM_POMPE_DA_COMANDARE *)
  AND( [ %MW9 = 3 ]       (* ORDINE_SECONDA_POMPA *)
  OR [ %MW9 = 0 ]         (* ORDINE_SECONDA_POMPA *)
  )
  AND %M4                 (* P3_USABILE *)
  ANDN %Q0.2              (* P3_CMD *)
  S %Q0.2                 (* P3_CMD *)
  [ %MW1 := %MW1 + 1 ]    (* NUM_POMPE_COMANDATE, NUM_POMPE_COMANDATE *)
  S %M12                  (* SECONDA_POMPA_COMANDATA *)
  // as ST:
  //   _t1 := NUM_POMPE_COMANDATE < NUM_POMPE_DA_COMANDARE AND NUM_POMPE_DA_COMANDARE >= 2 AND (ORDINE_SECONDA_POMPA = 3 OR ORDINE_SECONDA_POMPA = 0) AND P3_USABILE AND NOT P3_CMD;
  //   IF _t1 THEN P3_CMD := TRUE; END_IF;
  //   IF _t1 THEN NUM_POMPE_COMANDATE := NUM_POMPE_COMANDATE + 1; END_IF;
  //   IF _t1 THEN SECONDA_POMPA_COMANDATA := TRUE; END_IF;

// Rung 52
// Comanda: Seconda Pompa (Pompa 4)
  LD [ %MW1 < %MW0 ]      (* NUM_POMPE_COMANDATE, NUM_POMPE_DA_COMANDARE *)
  AND [ %MW0 >= 2 ]       (* NUM_POMPE_DA_COMANDARE *)
  AND( [ %MW9 = 4 ]       (* ORDINE_SECONDA_POMPA *)
  OR [ %MW9 = 0 ]         (* ORDINE_SECONDA_POMPA *)
  )
  AND %M5                 (* P4_USABILE *)
  ANDN %Q0.3              (* P4_CMD *)
  S %Q0.3                 (* P4_CMD *)
  [ %MW1 := %MW1 + 1 ]    (* NUM_POMPE_COMANDATE, NUM_POMPE_COMANDATE *)
  S %M12                  (* SECONDA_POMPA_COMANDATA *)
  // as ST:
  //   _t1 := NUM_POMPE_COMANDATE < NUM_POMPE_DA_COMANDARE AND NUM_POMPE_DA_COMANDARE >= 2 AND (ORDINE_SECONDA_POMPA = 4 OR ORDINE_SECONDA_POMPA = 0) AND P4_USABILE AND NOT P4_CMD;
  //   IF _t1 THEN P4_CMD := TRUE; END_IF;
  //   IF _t1 THEN NUM_POMPE_COMANDATE := NUM_POMPE_COMANDATE + 1; END_IF;
  //   IF _t1 THEN SECONDA_POMPA_COMANDATA := TRUE; END_IF;

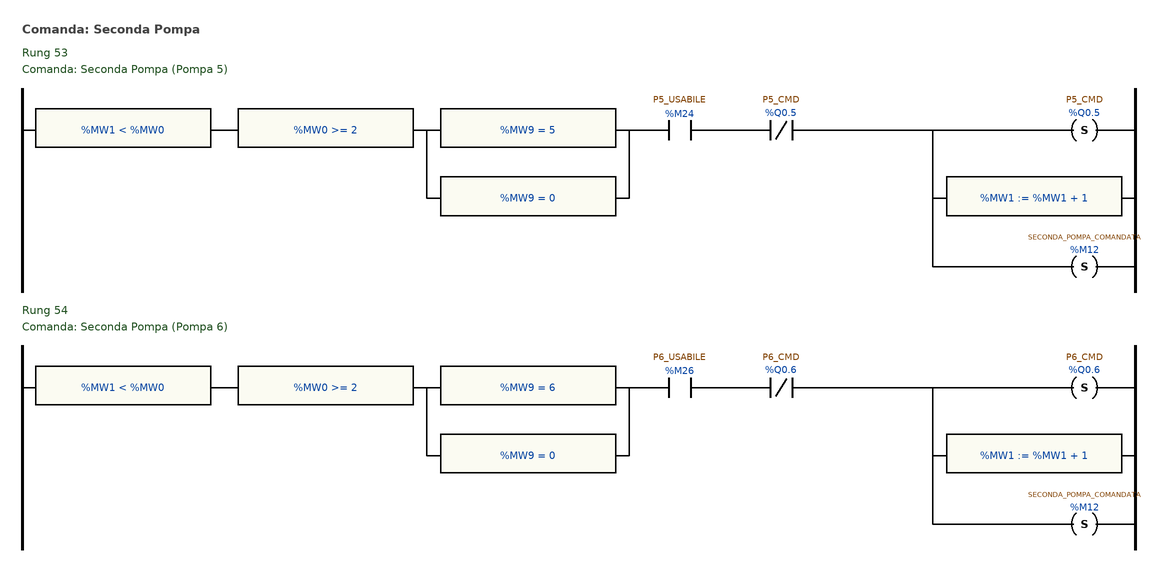

// Rung 53
// Comanda: Seconda Pompa (Pompa 5)
  LD [ %MW1 < %MW0 ]      (* NUM_POMPE_COMANDATE, NUM_POMPE_DA_COMANDARE *)
  AND [ %MW0 >= 2 ]       (* NUM_POMPE_DA_COMANDARE *)
  AND( [ %MW9 = 5 ]       (* ORDINE_SECONDA_POMPA *)
  OR [ %MW9 = 0 ]         (* ORDINE_SECONDA_POMPA *)
  )
  AND %M24                (* P5_USABILE *)
  ANDN %Q0.5              (* P5_CMD *)
  S %Q0.5                 (* P5_CMD *)
  [ %MW1 := %MW1 + 1 ]    (* NUM_POMPE_COMANDATE, NUM_POMPE_COMANDATE *)
  S %M12                  (* SECONDA_POMPA_COMANDATA *)
  // as ST:
  //   _t1 := NUM_POMPE_COMANDATE < NUM_POMPE_DA_COMANDARE AND NUM_POMPE_DA_COMANDARE >= 2 AND (ORDINE_SECONDA_POMPA = 5 OR ORDINE_SECONDA_POMPA = 0) AND P5_USABILE AND NOT P5_CMD;
  //   IF _t1 THEN P5_CMD := TRUE; END_IF;
  //   IF _t1 THEN NUM_POMPE_COMANDATE := NUM_POMPE_COMANDATE + 1; END_IF;
  //   IF _t1 THEN SECONDA_POMPA_COMANDATA := TRUE; END_IF;

// Rung 54
// Comanda: Seconda Pompa (Pompa 6)
  LD [ %MW1 < %MW0 ]      (* NUM_POMPE_COMANDATE, NUM_POMPE_DA_COMANDARE *)
  AND [ %MW0 >= 2 ]       (* NUM_POMPE_DA_COMANDARE *)
  AND( [ %MW9 = 6 ]       (* ORDINE_SECONDA_POMPA *)
  OR [ %MW9 = 0 ]         (* ORDINE_SECONDA_POMPA *)
  )
  AND %M26                (* P6_USABILE *)
  ANDN %Q0.6              (* P6_CMD *)
  S %Q0.6                 (* P6_CMD *)
  [ %MW1 := %MW1 + 1 ]    (* NUM_POMPE_COMANDATE, NUM_POMPE_COMANDATE *)
  S %M12                  (* SECONDA_POMPA_COMANDATA *)
  // as ST:
  //   _t1 := NUM_POMPE_COMANDATE < NUM_POMPE_DA_COMANDARE AND NUM_POMPE_DA_COMANDARE >= 2 AND (ORDINE_SECONDA_POMPA = 6 OR ORDINE_SECONDA_POMPA = 0) AND P6_USABILE AND NOT P6_CMD;
  //   IF _t1 THEN P6_CMD := TRUE; END_IF;
  //   IF _t1 THEN NUM_POMPE_COMANDATE := NUM_POMPE_COMANDATE + 1; END_IF;
  //   IF _t1 THEN SECONDA_POMPA_COMANDATA := TRUE; END_IF;

Subroutine Comanda: Terza Pompa
  (* SectionNumber=7, Number=5 *)

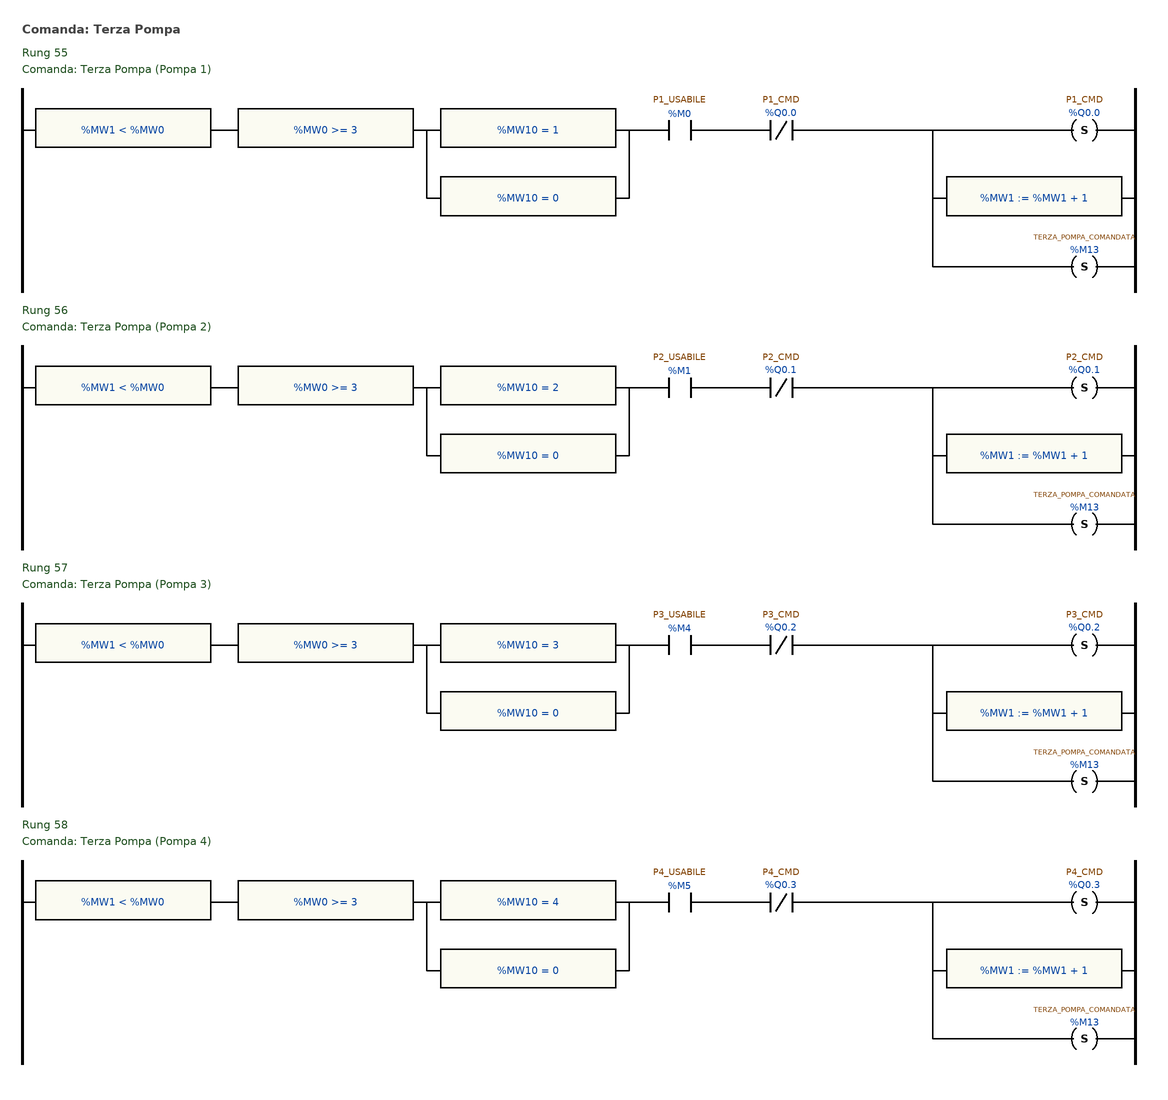

// Rung 55
// Comanda: Terza Pompa (Pompa 1)
  LD [ %MW1 < %MW0 ]      (* NUM_POMPE_COMANDATE, NUM_POMPE_DA_COMANDARE *)
  AND [ %MW0 >= 3 ]       (* NUM_POMPE_DA_COMANDARE *)
  AND( [ %MW10 = 1 ]      (* ORDINE_TERZA_POMPA *)
  OR [ %MW10 = 0 ]        (* ORDINE_TERZA_POMPA *)
  )
  AND %M0                 (* P1_USABILE *)
  ANDN %Q0.0              (* P1_CMD *)
  S %Q0.0                 (* P1_CMD *)
  [ %MW1 := %MW1 + 1 ]    (* NUM_POMPE_COMANDATE, NUM_POMPE_COMANDATE *)
  S %M13                  (* TERZA_POMPA_COMANDATA *)
  // as ST:
  //   _t1 := NUM_POMPE_COMANDATE < NUM_POMPE_DA_COMANDARE AND NUM_POMPE_DA_COMANDARE >= 3 AND (ORDINE_TERZA_POMPA = 1 OR ORDINE_TERZA_POMPA = 0) AND P1_USABILE AND NOT P1_CMD;
  //   IF _t1 THEN P1_CMD := TRUE; END_IF;
  //   IF _t1 THEN NUM_POMPE_COMANDATE := NUM_POMPE_COMANDATE + 1; END_IF;
  //   IF _t1 THEN TERZA_POMPA_COMANDATA := TRUE; END_IF;

// Rung 56
// Comanda: Terza Pompa (Pompa 2)
  LD [ %MW1 < %MW0 ]      (* NUM_POMPE_COMANDATE, NUM_POMPE_DA_COMANDARE *)
  AND [ %MW0 >= 3 ]       (* NUM_POMPE_DA_COMANDARE *)
  AND( [ %MW10 = 2 ]      (* ORDINE_TERZA_POMPA *)
  OR [ %MW10 = 0 ]        (* ORDINE_TERZA_POMPA *)
  )
  AND %M1                 (* P2_USABILE *)
  ANDN %Q0.1              (* P2_CMD *)
  S %Q0.1                 (* P2_CMD *)
  [ %MW1 := %MW1 + 1 ]    (* NUM_POMPE_COMANDATE, NUM_POMPE_COMANDATE *)
  S %M13                  (* TERZA_POMPA_COMANDATA *)
  // as ST:
  //   _t1 := NUM_POMPE_COMANDATE < NUM_POMPE_DA_COMANDARE AND NUM_POMPE_DA_COMANDARE >= 3 AND (ORDINE_TERZA_POMPA = 2 OR ORDINE_TERZA_POMPA = 0) AND P2_USABILE AND NOT P2_CMD;
  //   IF _t1 THEN P2_CMD := TRUE; END_IF;
  //   IF _t1 THEN NUM_POMPE_COMANDATE := NUM_POMPE_COMANDATE + 1; END_IF;
  //   IF _t1 THEN TERZA_POMPA_COMANDATA := TRUE; END_IF;

// Rung 57
// Comanda: Terza Pompa (Pompa 3)
  LD [ %MW1 < %MW0 ]      (* NUM_POMPE_COMANDATE, NUM_POMPE_DA_COMANDARE *)
  AND [ %MW0 >= 3 ]       (* NUM_POMPE_DA_COMANDARE *)
  AND( [ %MW10 = 3 ]      (* ORDINE_TERZA_POMPA *)
  OR [ %MW10 = 0 ]        (* ORDINE_TERZA_POMPA *)
  )
  AND %M4                 (* P3_USABILE *)
  ANDN %Q0.2              (* P3_CMD *)
  S %Q0.2                 (* P3_CMD *)
  [ %MW1 := %MW1 + 1 ]    (* NUM_POMPE_COMANDATE, NUM_POMPE_COMANDATE *)
  S %M13                  (* TERZA_POMPA_COMANDATA *)
  // as ST:
  //   _t1 := NUM_POMPE_COMANDATE < NUM_POMPE_DA_COMANDARE AND NUM_POMPE_DA_COMANDARE >= 3 AND (ORDINE_TERZA_POMPA = 3 OR ORDINE_TERZA_POMPA = 0) AND P3_USABILE AND NOT P3_CMD;
  //   IF _t1 THEN P3_CMD := TRUE; END_IF;
  //   IF _t1 THEN NUM_POMPE_COMANDATE := NUM_POMPE_COMANDATE + 1; END_IF;
  //   IF _t1 THEN TERZA_POMPA_COMANDATA := TRUE; END_IF;

// Rung 58
// Comanda: Terza Pompa (Pompa 4)
  LD [ %MW1 < %MW0 ]      (* NUM_POMPE_COMANDATE, NUM_POMPE_DA_COMANDARE *)
  AND [ %MW0 >= 3 ]       (* NUM_POMPE_DA_COMANDARE *)
  AND( [ %MW10 = 4 ]      (* ORDINE_TERZA_POMPA *)
  OR [ %MW10 = 0 ]        (* ORDINE_TERZA_POMPA *)
  )
  AND %M5                 (* P4_USABILE *)
  ANDN %Q0.3              (* P4_CMD *)
  S %Q0.3                 (* P4_CMD *)
  [ %MW1 := %MW1 + 1 ]    (* NUM_POMPE_COMANDATE, NUM_POMPE_COMANDATE *)
  S %M13                  (* TERZA_POMPA_COMANDATA *)
  // as ST:
  //   _t1 := NUM_POMPE_COMANDATE < NUM_POMPE_DA_COMANDARE AND NUM_POMPE_DA_COMANDARE >= 3 AND (ORDINE_TERZA_POMPA = 4 OR ORDINE_TERZA_POMPA = 0) AND P4_USABILE AND NOT P4_CMD;
  //   IF _t1 THEN P4_CMD := TRUE; END_IF;
  //   IF _t1 THEN NUM_POMPE_COMANDATE := NUM_POMPE_COMANDATE + 1; END_IF;
  //   IF _t1 THEN TERZA_POMPA_COMANDATA := TRUE; END_IF;

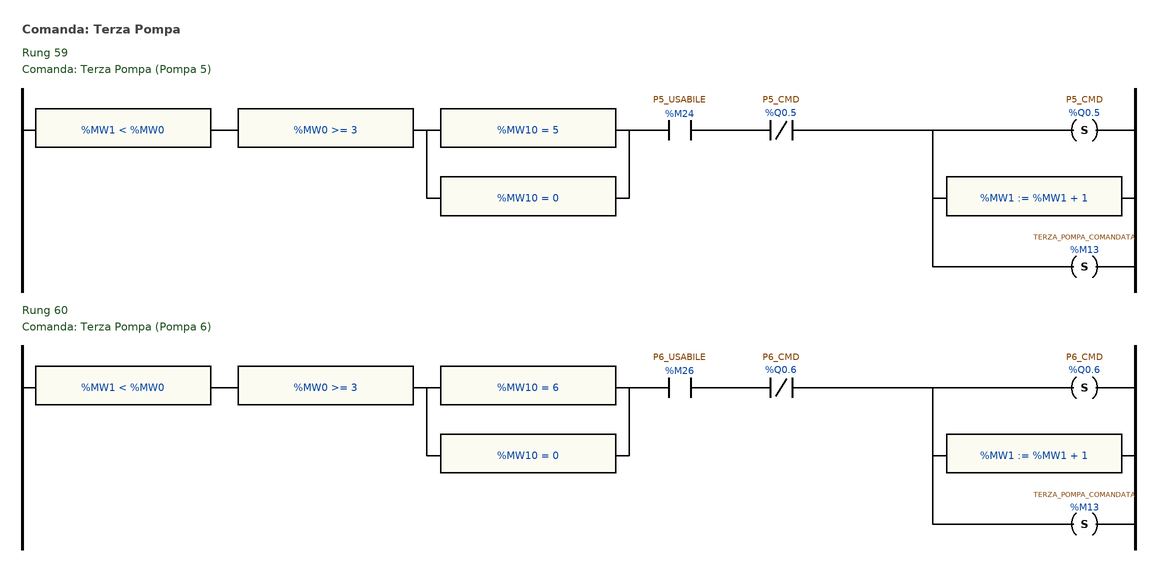

// Rung 59
// Comanda: Terza Pompa (Pompa 5)
  LD [ %MW1 < %MW0 ]      (* NUM_POMPE_COMANDATE, NUM_POMPE_DA_COMANDARE *)
  AND [ %MW0 >= 3 ]       (* NUM_POMPE_DA_COMANDARE *)
  AND( [ %MW10 = 5 ]      (* ORDINE_TERZA_POMPA *)
  OR [ %MW10 = 0 ]        (* ORDINE_TERZA_POMPA *)
  )
  AND %M24                (* P5_USABILE *)
  ANDN %Q0.5              (* P5_CMD *)
  S %Q0.5                 (* P5_CMD *)
  [ %MW1 := %MW1 + 1 ]    (* NUM_POMPE_COMANDATE, NUM_POMPE_COMANDATE *)
  S %M13                  (* TERZA_POMPA_COMANDATA *)
  // as ST:
  //   _t1 := NUM_POMPE_COMANDATE < NUM_POMPE_DA_COMANDARE AND NUM_POMPE_DA_COMANDARE >= 3 AND (ORDINE_TERZA_POMPA = 5 OR ORDINE_TERZA_POMPA = 0) AND P5_USABILE AND NOT P5_CMD;
  //   IF _t1 THEN P5_CMD := TRUE; END_IF;
  //   IF _t1 THEN NUM_POMPE_COMANDATE := NUM_POMPE_COMANDATE + 1; END_IF;
  //   IF _t1 THEN TERZA_POMPA_COMANDATA := TRUE; END_IF;

// Rung 60
// Comanda: Terza Pompa (Pompa 6)
  LD [ %MW1 < %MW0 ]      (* NUM_POMPE_COMANDATE, NUM_POMPE_DA_COMANDARE *)
  AND [ %MW0 >= 3 ]       (* NUM_POMPE_DA_COMANDARE *)
  AND( [ %MW10 = 6 ]      (* ORDINE_TERZA_POMPA *)
  OR [ %MW10 = 0 ]        (* ORDINE_TERZA_POMPA *)
  )
  AND %M26                (* P6_USABILE *)
  ANDN %Q0.6              (* P6_CMD *)
  S %Q0.6                 (* P6_CMD *)
  [ %MW1 := %MW1 + 1 ]    (* NUM_POMPE_COMANDATE, NUM_POMPE_COMANDATE *)
  S %M13                  (* TERZA_POMPA_COMANDATA *)
  // as ST:
  //   _t1 := NUM_POMPE_COMANDATE < NUM_POMPE_DA_COMANDARE AND NUM_POMPE_DA_COMANDARE >= 3 AND (ORDINE_TERZA_POMPA = 6 OR ORDINE_TERZA_POMPA = 0) AND P6_USABILE AND NOT P6_CMD;
  //   IF _t1 THEN P6_CMD := TRUE; END_IF;
  //   IF _t1 THEN NUM_POMPE_COMANDATE := NUM_POMPE_COMANDATE + 1; END_IF;
  //   IF _t1 THEN TERZA_POMPA_COMANDATA := TRUE; END_IF;

Subroutine Conta Secondi per Pompa
  (* SectionNumber=8, Number=6 *)

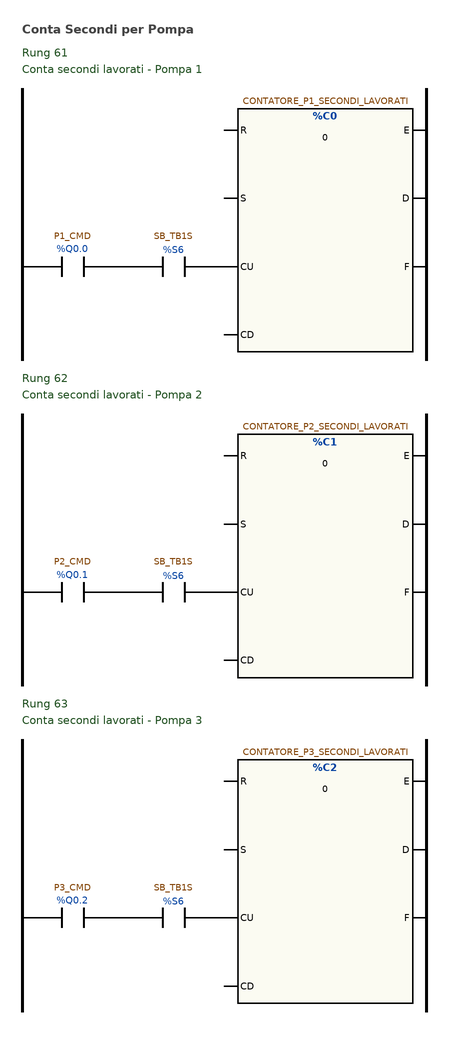

// Rung 61
// Conta secondi lavorati - Pompa 1
  BLK %C0                 (* CONTATORE_P1_SECONDI_LAVORATI *)
  LD %Q0.0                (* P1_CMD *)
  AND %S6                 (* SB_TB1S *)
  CU
  END_BLK
  // as ST:
  //   CONTATORE_P1_SECONDI_LAVORATI(CU := P1_CMD AND SB_TB1S);

// Rung 62
// Conta secondi lavorati - Pompa 2
  BLK %C1                 (* CONTATORE_P2_SECONDI_LAVORATI *)
  LD %Q0.1                (* P2_CMD *)
  AND %S6                 (* SB_TB1S *)
  CU
  END_BLK
  // as ST:
  //   CONTATORE_P2_SECONDI_LAVORATI(CU := P2_CMD AND SB_TB1S);

// Rung 63
// Conta secondi lavorati - Pompa 3
  BLK %C2                 (* CONTATORE_P3_SECONDI_LAVORATI *)
  LD %Q0.2                (* P3_CMD *)
  AND %S6                 (* SB_TB1S *)
  CU
  END_BLK
  // as ST:
  //   CONTATORE_P3_SECONDI_LAVORATI(CU := P3_CMD AND SB_TB1S);

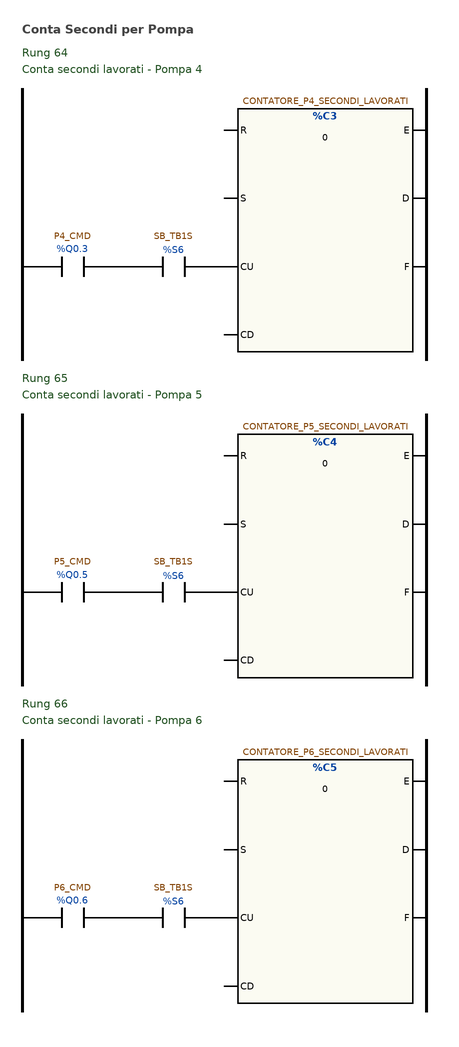

// Rung 64
// Conta secondi lavorati - Pompa 4
  BLK %C3                 (* CONTATORE_P4_SECONDI_LAVORATI *)
  LD %Q0.3                (* P4_CMD *)
  AND %S6                 (* SB_TB1S *)
  CU
  END_BLK
  // as ST:
  //   CONTATORE_P4_SECONDI_LAVORATI(CU := P4_CMD AND SB_TB1S);

// Rung 65
// Conta secondi lavorati - Pompa 5
  BLK %C4                 (* CONTATORE_P5_SECONDI_LAVORATI *)
  LD %Q0.5                (* P5_CMD *)
  AND %S6                 (* SB_TB1S *)
  CU
  END_BLK
  // as ST:
  //   CONTATORE_P5_SECONDI_LAVORATI(CU := P5_CMD AND SB_TB1S);

// Rung 66
// Conta secondi lavorati - Pompa 6
  BLK %C5                 (* CONTATORE_P6_SECONDI_LAVORATI *)
  LD %Q0.6                (* P6_CMD *)
  AND %S6                 (* SB_TB1S *)
  CU
  END_BLK
  // as ST:
  //   CONTATORE_P6_SECONDI_LAVORATI(CU := P6_CMD AND SB_TB1S);

Subroutine Disattivazione Pompe 
  (* SectionNumber=9, Number=7 *)

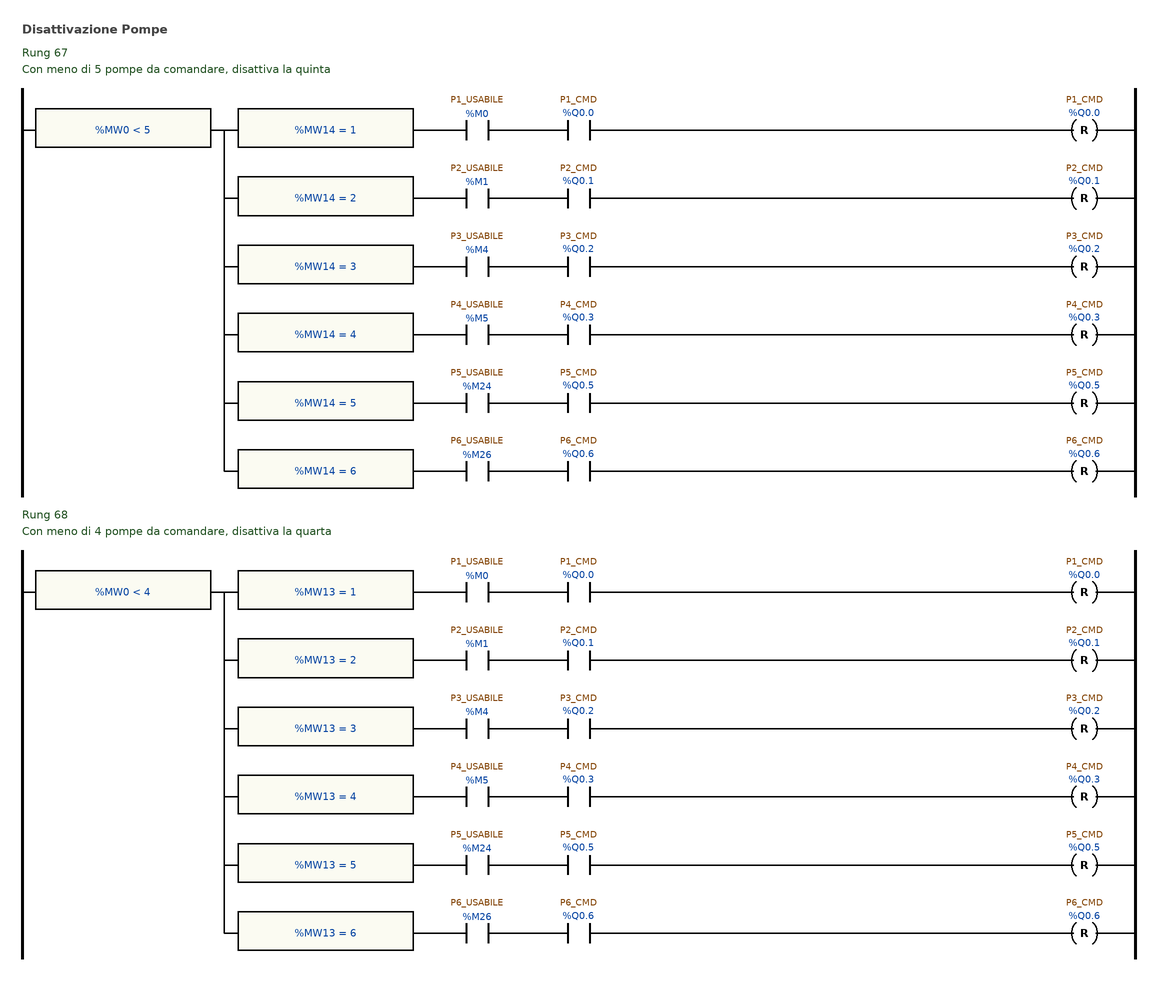

// Rung 67
// Con meno di 5 pompe da comandare, disattiva la quinta
  LD [ %MW0 < 5 ]         (* NUM_POMPE_DA_COMANDARE *)
  MPS
  AND [ %MW14 = 1 ]       (* ORDINE_QUINTA_POMPA *)
  AND %M0                 (* P1_USABILE *)
  AND %Q0.0               (* P1_CMD *)
  R %Q0.0                 (* P1_CMD *)
  MRD
  AND [ %MW14 = 2 ]       (* ORDINE_QUINTA_POMPA *)
  AND %M1                 (* P2_USABILE *)
  AND %Q0.1               (* P2_CMD *)
  R %Q0.1                 (* P2_CMD *)
  MRD
  AND [ %MW14 = 3 ]       (* ORDINE_QUINTA_POMPA *)
  AND %M4                 (* P3_USABILE *)
  AND %Q0.2               (* P3_CMD *)
  R %Q0.2                 (* P3_CMD *)
  MRD
  AND [ %MW14 = 4 ]       (* ORDINE_QUINTA_POMPA *)
  AND %M5                 (* P4_USABILE *)
  AND %Q0.3               (* P4_CMD *)
  R %Q0.3                 (* P4_CMD *)
  MRD
  AND [ %MW14 = 5 ]       (* ORDINE_QUINTA_POMPA *)
  AND %M24                (* P5_USABILE *)
  AND %Q0.5               (* P5_CMD *)
  R %Q0.5                 (* P5_CMD *)
  MPP
  AND [ %MW14 = 6 ]       (* ORDINE_QUINTA_POMPA *)
  AND %M26                (* P6_USABILE *)
  AND %Q0.6               (* P6_CMD *)
  R %Q0.6                 (* P6_CMD *)
  // as ST:
  //   IF NUM_POMPE_DA_COMANDARE < 5 AND ORDINE_QUINTA_POMPA = 1 AND P1_USABILE AND P1_CMD THEN P1_CMD := FALSE; END_IF;
  //   IF NUM_POMPE_DA_COMANDARE < 5 AND ORDINE_QUINTA_POMPA = 2 AND P2_USABILE AND P2_CMD THEN P2_CMD := FALSE; END_IF;
  //   IF NUM_POMPE_DA_COMANDARE < 5 AND ORDINE_QUINTA_POMPA = 3 AND P3_USABILE AND P3_CMD THEN P3_CMD := FALSE; END_IF;
  //   IF NUM_POMPE_DA_COMANDARE < 5 AND ORDINE_QUINTA_POMPA = 4 AND P4_USABILE AND P4_CMD THEN P4_CMD := FALSE; END_IF;
  //   IF NUM_POMPE_DA_COMANDARE < 5 AND ORDINE_QUINTA_POMPA = 5 AND P5_USABILE AND P5_CMD THEN P5_CMD := FALSE; END_IF;
  //   IF NUM_POMPE_DA_COMANDARE < 5 AND ORDINE_QUINTA_POMPA = 6 AND P6_USABILE AND P6_CMD THEN P6_CMD := FALSE; END_IF;

// Rung 68
// Con meno di 4 pompe da comandare, disattiva la quarta
  LD [ %MW0 < 4 ]         (* NUM_POMPE_DA_COMANDARE *)
  MPS
  AND [ %MW13 = 1 ]       (* ORDINE_QUARTA_POMPA *)
  AND %M0                 (* P1_USABILE *)
  AND %Q0.0               (* P1_CMD *)
  R %Q0.0                 (* P1_CMD *)
  MRD
  AND [ %MW13 = 2 ]       (* ORDINE_QUARTA_POMPA *)
  AND %M1                 (* P2_USABILE *)
  AND %Q0.1               (* P2_CMD *)
  R %Q0.1                 (* P2_CMD *)
  MRD
  AND [ %MW13 = 3 ]       (* ORDINE_QUARTA_POMPA *)
  AND %M4                 (* P3_USABILE *)
  AND %Q0.2               (* P3_CMD *)
  R %Q0.2                 (* P3_CMD *)
  MRD
  AND [ %MW13 = 4 ]       (* ORDINE_QUARTA_POMPA *)
  AND %M5                 (* P4_USABILE *)
  AND %Q0.3               (* P4_CMD *)
  R %Q0.3                 (* P4_CMD *)
  MRD
  AND [ %MW13 = 5 ]       (* ORDINE_QUARTA_POMPA *)
  AND %M24                (* P5_USABILE *)
  AND %Q0.5               (* P5_CMD *)
  R %Q0.5                 (* P5_CMD *)
  MPP
  AND [ %MW13 = 6 ]       (* ORDINE_QUARTA_POMPA *)
  AND %M26                (* P6_USABILE *)
  AND %Q0.6               (* P6_CMD *)
  R %Q0.6                 (* P6_CMD *)
  // as ST:
  //   IF NUM_POMPE_DA_COMANDARE < 4 AND ORDINE_QUARTA_POMPA = 1 AND P1_USABILE AND P1_CMD THEN P1_CMD := FALSE; END_IF;
  //   IF NUM_POMPE_DA_COMANDARE < 4 AND ORDINE_QUARTA_POMPA = 2 AND P2_USABILE AND P2_CMD THEN P2_CMD := FALSE; END_IF;
  //   IF NUM_POMPE_DA_COMANDARE < 4 AND ORDINE_QUARTA_POMPA = 3 AND P3_USABILE AND P3_CMD THEN P3_CMD := FALSE; END_IF;
  //   IF NUM_POMPE_DA_COMANDARE < 4 AND ORDINE_QUARTA_POMPA = 4 AND P4_USABILE AND P4_CMD THEN P4_CMD := FALSE; END_IF;
  //   IF NUM_POMPE_DA_COMANDARE < 4 AND ORDINE_QUARTA_POMPA = 5 AND P5_USABILE AND P5_CMD THEN P5_CMD := FALSE; END_IF;
  //   IF NUM_POMPE_DA_COMANDARE < 4 AND ORDINE_QUARTA_POMPA = 6 AND P6_USABILE AND P6_CMD THEN P6_CMD := FALSE; END_IF;

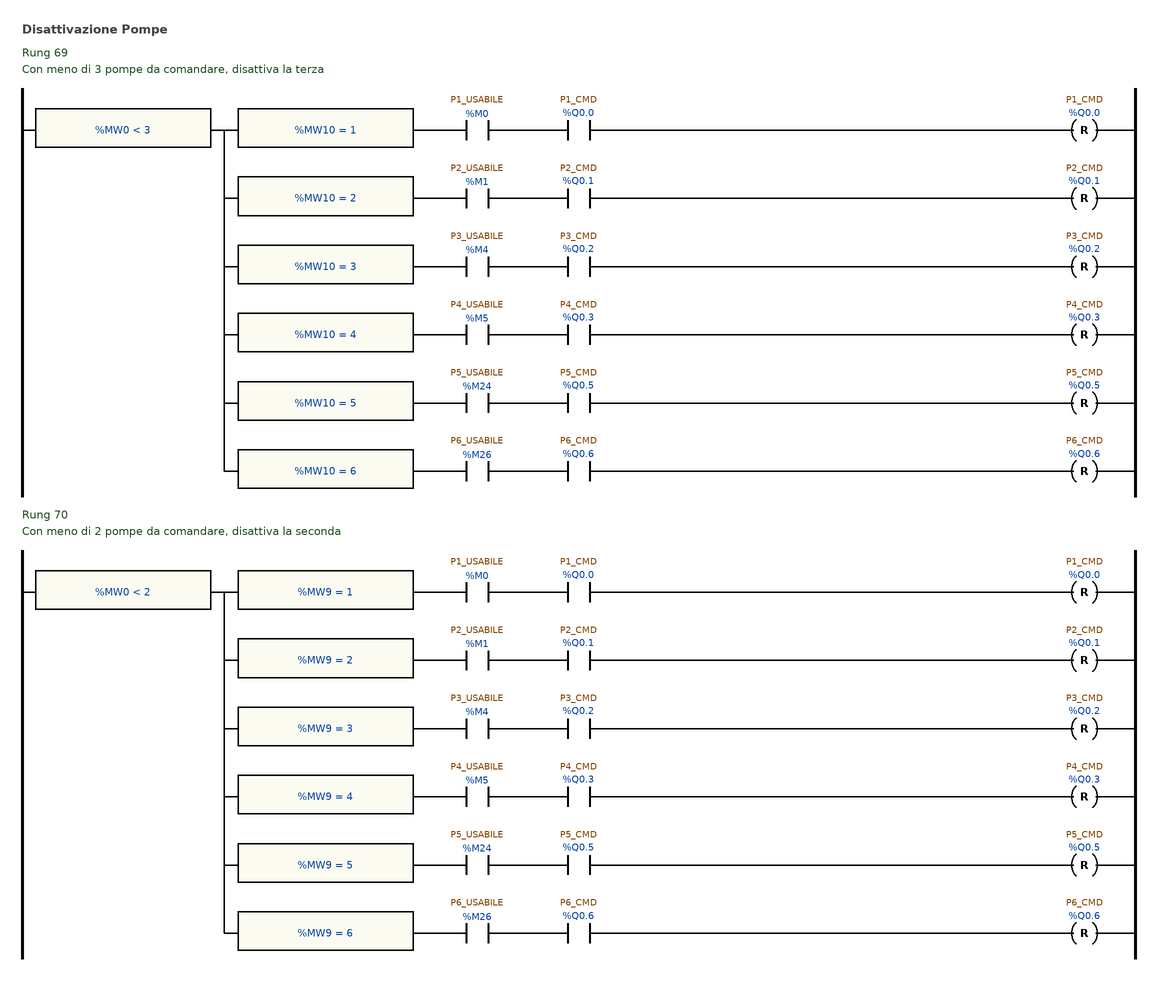

// Rung 69
// Con meno di 3 pompe da comandare, disattiva la terza
  LD [ %MW0 < 3 ]         (* NUM_POMPE_DA_COMANDARE *)
  MPS
  AND [ %MW10 = 1 ]       (* ORDINE_TERZA_POMPA *)
  AND %M0                 (* P1_USABILE *)
  AND %Q0.0               (* P1_CMD *)
  R %Q0.0                 (* P1_CMD *)
  MRD
  AND [ %MW10 = 2 ]       (* ORDINE_TERZA_POMPA *)
  AND %M1                 (* P2_USABILE *)
  AND %Q0.1               (* P2_CMD *)
  R %Q0.1                 (* P2_CMD *)
  MRD
  AND [ %MW10 = 3 ]       (* ORDINE_TERZA_POMPA *)
  AND %M4                 (* P3_USABILE *)
  AND %Q0.2               (* P3_CMD *)
  R %Q0.2                 (* P3_CMD *)
  MRD
  AND [ %MW10 = 4 ]       (* ORDINE_TERZA_POMPA *)
  AND %M5                 (* P4_USABILE *)
  AND %Q0.3               (* P4_CMD *)
  R %Q0.3                 (* P4_CMD *)
  MRD
  AND [ %MW10 = 5 ]       (* ORDINE_TERZA_POMPA *)
  AND %M24                (* P5_USABILE *)
  AND %Q0.5               (* P5_CMD *)
  R %Q0.5                 (* P5_CMD *)
  MPP
  AND [ %MW10 = 6 ]       (* ORDINE_TERZA_POMPA *)
  AND %M26                (* P6_USABILE *)
  AND %Q0.6               (* P6_CMD *)
  R %Q0.6                 (* P6_CMD *)
  // as ST:
  //   IF NUM_POMPE_DA_COMANDARE < 3 AND ORDINE_TERZA_POMPA = 1 AND P1_USABILE AND P1_CMD THEN P1_CMD := FALSE; END_IF;
  //   IF NUM_POMPE_DA_COMANDARE < 3 AND ORDINE_TERZA_POMPA = 2 AND P2_USABILE AND P2_CMD THEN P2_CMD := FALSE; END_IF;
  //   IF NUM_POMPE_DA_COMANDARE < 3 AND ORDINE_TERZA_POMPA = 3 AND P3_USABILE AND P3_CMD THEN P3_CMD := FALSE; END_IF;
  //   IF NUM_POMPE_DA_COMANDARE < 3 AND ORDINE_TERZA_POMPA = 4 AND P4_USABILE AND P4_CMD THEN P4_CMD := FALSE; END_IF;
  //   IF NUM_POMPE_DA_COMANDARE < 3 AND ORDINE_TERZA_POMPA = 5 AND P5_USABILE AND P5_CMD THEN P5_CMD := FALSE; END_IF;
  //   IF NUM_POMPE_DA_COMANDARE < 3 AND ORDINE_TERZA_POMPA = 6 AND P6_USABILE AND P6_CMD THEN P6_CMD := FALSE; END_IF;

// Rung 70
// Con meno di 2 pompe da comandare, disattiva la seconda
  LD [ %MW0 < 2 ]         (* NUM_POMPE_DA_COMANDARE *)
  MPS
  AND [ %MW9 = 1 ]        (* ORDINE_SECONDA_POMPA *)
  AND %M0                 (* P1_USABILE *)
  AND %Q0.0               (* P1_CMD *)
  R %Q0.0                 (* P1_CMD *)
  MRD
  AND [ %MW9 = 2 ]        (* ORDINE_SECONDA_POMPA *)
  AND %M1                 (* P2_USABILE *)
  AND %Q0.1               (* P2_CMD *)
  R %Q0.1                 (* P2_CMD *)
  MRD
  AND [ %MW9 = 3 ]        (* ORDINE_SECONDA_POMPA *)
  AND %M4                 (* P3_USABILE *)
  AND %Q0.2               (* P3_CMD *)
  R %Q0.2                 (* P3_CMD *)
  MRD
  AND [ %MW9 = 4 ]        (* ORDINE_SECONDA_POMPA *)
  AND %M5                 (* P4_USABILE *)
  AND %Q0.3               (* P4_CMD *)
  R %Q0.3                 (* P4_CMD *)
  MRD
  AND [ %MW9 = 5 ]        (* ORDINE_SECONDA_POMPA *)
  AND %M24                (* P5_USABILE *)
  AND %Q0.5               (* P5_CMD *)
  R %Q0.5                 (* P5_CMD *)
  MPP
  AND [ %MW9 = 6 ]        (* ORDINE_SECONDA_POMPA *)
  AND %M26                (* P6_USABILE *)
  AND %Q0.6               (* P6_CMD *)
  R %Q0.6                 (* P6_CMD *)
  // as ST:
  //   IF NUM_POMPE_DA_COMANDARE < 2 AND ORDINE_SECONDA_POMPA = 1 AND P1_USABILE AND P1_CMD THEN P1_CMD := FALSE; END_IF;
  //   IF NUM_POMPE_DA_COMANDARE < 2 AND ORDINE_SECONDA_POMPA = 2 AND P2_USABILE AND P2_CMD THEN P2_CMD := FALSE; END_IF;
  //   IF NUM_POMPE_DA_COMANDARE < 2 AND ORDINE_SECONDA_POMPA = 3 AND P3_USABILE AND P3_CMD THEN P3_CMD := FALSE; END_IF;
  //   IF NUM_POMPE_DA_COMANDARE < 2 AND ORDINE_SECONDA_POMPA = 4 AND P4_USABILE AND P4_CMD THEN P4_CMD := FALSE; END_IF;
  //   IF NUM_POMPE_DA_COMANDARE < 2 AND ORDINE_SECONDA_POMPA = 5 AND P5_USABILE AND P5_CMD THEN P5_CMD := FALSE; END_IF;
  //   IF NUM_POMPE_DA_COMANDARE < 2 AND ORDINE_SECONDA_POMPA = 6 AND P6_USABILE AND P6_CMD THEN P6_CMD := FALSE; END_IF;

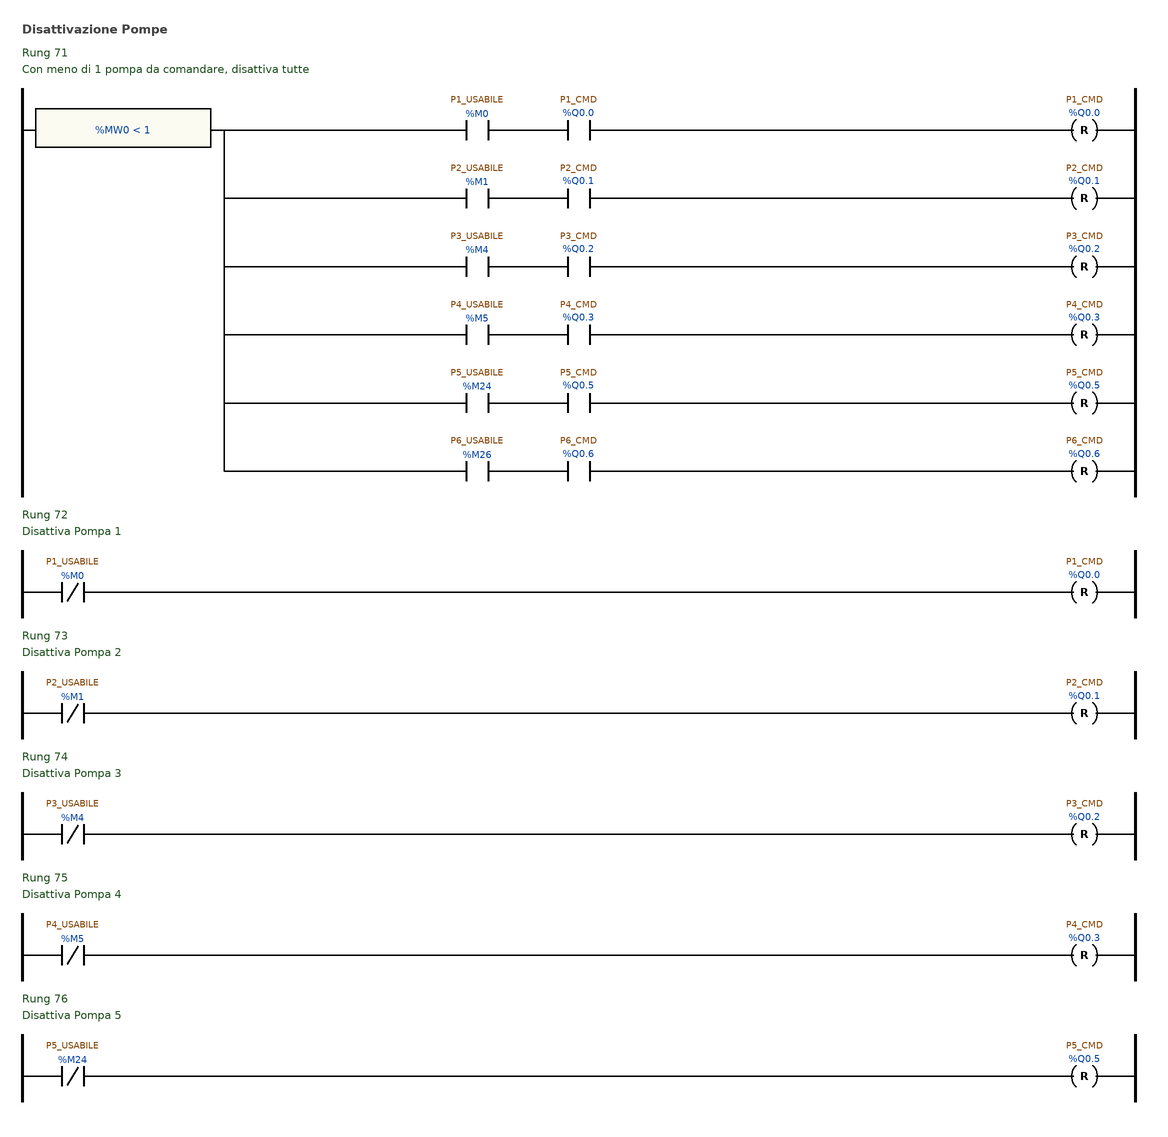

// Rung 71
// Con meno di 1 pompa da comandare, disattiva tutte
  LD [ %MW0 < 1 ]         (* NUM_POMPE_DA_COMANDARE *)
  MPS
  AND %M0                 (* P1_USABILE *)
  AND %Q0.0               (* P1_CMD *)
  R %Q0.0                 (* P1_CMD *)
  MRD
  AND %M1                 (* P2_USABILE *)
  AND %Q0.1               (* P2_CMD *)
  R %Q0.1                 (* P2_CMD *)
  MRD
  AND %M4                 (* P3_USABILE *)
  AND %Q0.2               (* P3_CMD *)
  R %Q0.2                 (* P3_CMD *)
  MRD
  AND %M5                 (* P4_USABILE *)
  AND %Q0.3               (* P4_CMD *)
  R %Q0.3                 (* P4_CMD *)
  MRD
  AND %M24                (* P5_USABILE *)
  AND %Q0.5               (* P5_CMD *)
  R %Q0.5                 (* P5_CMD *)
  MPP
  AND %M26                (* P6_USABILE *)
  AND %Q0.6               (* P6_CMD *)
  R %Q0.6                 (* P6_CMD *)
  // as ST:
  //   IF NUM_POMPE_DA_COMANDARE < 1 AND P1_USABILE AND P1_CMD THEN P1_CMD := FALSE; END_IF;
  //   IF NUM_POMPE_DA_COMANDARE < 1 AND P2_USABILE AND P2_CMD THEN P2_CMD := FALSE; END_IF;
  //   IF NUM_POMPE_DA_COMANDARE < 1 AND P3_USABILE AND P3_CMD THEN P3_CMD := FALSE; END_IF;
  //   IF NUM_POMPE_DA_COMANDARE < 1 AND P4_USABILE AND P4_CMD THEN P4_CMD := FALSE; END_IF;
  //   IF NUM_POMPE_DA_COMANDARE < 1 AND P5_USABILE AND P5_CMD THEN P5_CMD := FALSE; END_IF;
  //   IF NUM_POMPE_DA_COMANDARE < 1 AND P6_USABILE AND P6_CMD THEN P6_CMD := FALSE; END_IF;

// Rung 72
// Disattiva Pompa 1
  LDN %M0                 (* P1_USABILE *)
  R %Q0.0                 (* P1_CMD *)
  // as ST:
  //   IF NOT P1_USABILE THEN P1_CMD := FALSE; END_IF;

// Rung 73
// Disattiva Pompa 2
  LDN %M1                 (* P2_USABILE *)
  R %Q0.1                 (* P2_CMD *)
  // as ST:
  //   IF NOT P2_USABILE THEN P2_CMD := FALSE; END_IF;

// Rung 74
// Disattiva Pompa 3
  LDN %M4                 (* P3_USABILE *)
  R %Q0.2                 (* P3_CMD *)
  // as ST:
  //   IF NOT P3_USABILE THEN P3_CMD := FALSE; END_IF;

// Rung 75
// Disattiva Pompa 4
  LDN %M5                 (* P4_USABILE *)
  R %Q0.3                 (* P4_CMD *)
  // as ST:
  //   IF NOT P4_USABILE THEN P4_CMD := FALSE; END_IF;

// Rung 76
// Disattiva Pompa 5
  LDN %M24                (* P5_USABILE *)
  R %Q0.5                 (* P5_CMD *)
  // as ST:
  //   IF NOT P5_USABILE THEN P5_CMD := FALSE; END_IF;

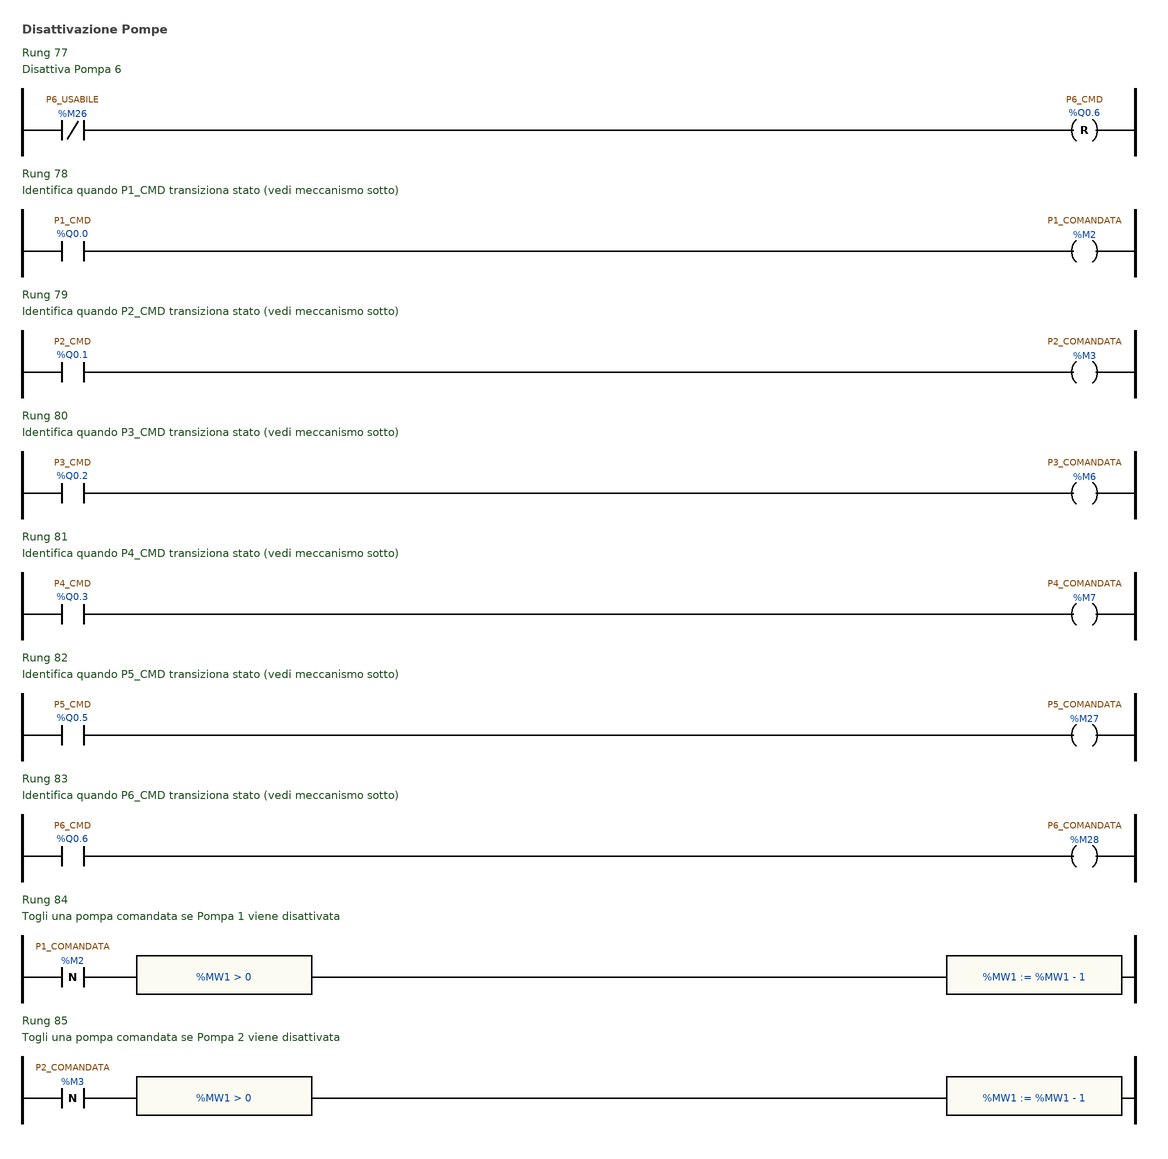

// Rung 77
// Disattiva Pompa 6
  LDN %M26                (* P6_USABILE *)
  R %Q0.6                 (* P6_CMD *)
  // as ST:
  //   IF NOT P6_USABILE THEN P6_CMD := FALSE; END_IF;

// Rung 78
// Identifica quando P1_CMD transiziona stato (vedi meccanismo sotto)
  LD %Q0.0                (* P1_CMD *)
  ST %M2                  (* P1_COMANDATA *)
  // as ST:
  //   P1_COMANDATA := P1_CMD;

// Rung 79
// Identifica quando P2_CMD transiziona stato (vedi meccanismo sotto)
  LD %Q0.1                (* P2_CMD *)
  ST %M3                  (* P2_COMANDATA *)
  // as ST:
  //   P2_COMANDATA := P2_CMD;

// Rung 80
// Identifica quando P3_CMD transiziona stato (vedi meccanismo sotto)
  LD %Q0.2                (* P3_CMD *)
  ST %M6                  (* P3_COMANDATA *)
  // as ST:
  //   P3_COMANDATA := P3_CMD;

// Rung 81
// Identifica quando P4_CMD transiziona stato (vedi meccanismo sotto)
  LD %Q0.3                (* P4_CMD *)
  ST %M7                  (* P4_COMANDATA *)
  // as ST:
  //   P4_COMANDATA := P4_CMD;

// Rung 82
// Identifica quando P5_CMD transiziona stato (vedi meccanismo sotto)
  LD %Q0.5                (* P5_CMD *)
  ST %M27                 (* P5_COMANDATA *)
  // as ST:
  //   P5_COMANDATA := P5_CMD;

// Rung 83
// Identifica quando P6_CMD transiziona stato (vedi meccanismo sotto)
  LD %Q0.6                (* P6_CMD *)
  ST %M28                 (* P6_COMANDATA *)
  // as ST:
  //   P6_COMANDATA := P6_CMD;

// Rung 84
// Togli una pompa comandata se Pompa 1 viene disattivata
  LDF %M2                 (* P1_COMANDATA *)
  AND [ %MW1 > 0 ]        (* NUM_POMPE_COMANDATE *)
  [ %MW1 := %MW1 - 1 ]    (* NUM_POMPE_COMANDATE, NUM_POMPE_COMANDATE *)
  // as ST:
  //   IF FALLING(P1_COMANDATA) AND NUM_POMPE_COMANDATE > 0 THEN NUM_POMPE_COMANDATE := NUM_POMPE_COMANDATE - 1; END_IF;

// Rung 85
// Togli una pompa comandata se Pompa 2 viene disattivata
  LDF %M3                 (* P2_COMANDATA *)
  AND [ %MW1 > 0 ]        (* NUM_POMPE_COMANDATE *)
  [ %MW1 := %MW1 - 1 ]    (* NUM_POMPE_COMANDATE, NUM_POMPE_COMANDATE *)
  // as ST:
  //   IF FALLING(P2_COMANDATA) AND NUM_POMPE_COMANDATE > 0 THEN NUM_POMPE_COMANDATE := NUM_POMPE_COMANDATE - 1; END_IF;

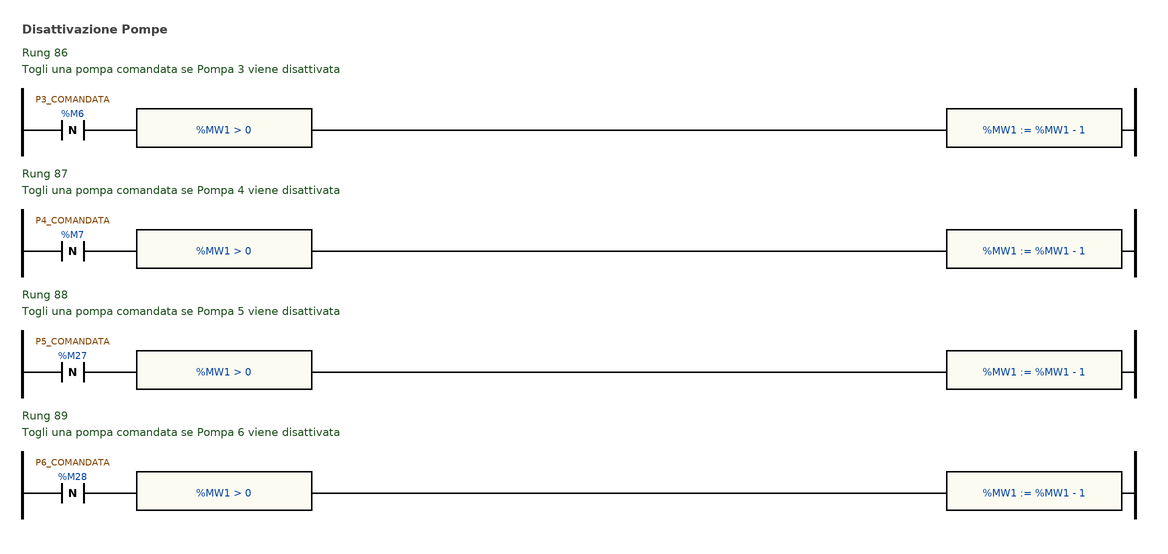

// Rung 86
// Togli una pompa comandata se Pompa 3 viene disattivata
  LDF %M6                 (* P3_COMANDATA *)
  AND [ %MW1 > 0 ]        (* NUM_POMPE_COMANDATE *)
  [ %MW1 := %MW1 - 1 ]    (* NUM_POMPE_COMANDATE, NUM_POMPE_COMANDATE *)
  // as ST:
  //   IF FALLING(P3_COMANDATA) AND NUM_POMPE_COMANDATE > 0 THEN NUM_POMPE_COMANDATE := NUM_POMPE_COMANDATE - 1; END_IF;

// Rung 87
// Togli una pompa comandata se Pompa 4 viene disattivata
  LDF %M7                 (* P4_COMANDATA *)
  AND [ %MW1 > 0 ]        (* NUM_POMPE_COMANDATE *)
  [ %MW1 := %MW1 - 1 ]    (* NUM_POMPE_COMANDATE, NUM_POMPE_COMANDATE *)
  // as ST:
  //   IF FALLING(P4_COMANDATA) AND NUM_POMPE_COMANDATE > 0 THEN NUM_POMPE_COMANDATE := NUM_POMPE_COMANDATE - 1; END_IF;

// Rung 88
// Togli una pompa comandata se Pompa 5 viene disattivata
  LDF %M27                (* P5_COMANDATA *)
  AND [ %MW1 > 0 ]        (* NUM_POMPE_COMANDATE *)
  [ %MW1 := %MW1 - 1 ]    (* NUM_POMPE_COMANDATE, NUM_POMPE_COMANDATE *)
  // as ST:
  //   IF FALLING(P5_COMANDATA) AND NUM_POMPE_COMANDATE > 0 THEN NUM_POMPE_COMANDATE := NUM_POMPE_COMANDATE - 1; END_IF;

// Rung 89
// Togli una pompa comandata se Pompa 6 viene disattivata
  LDF %M28                (* P6_COMANDATA *)
  AND [ %MW1 > 0 ]        (* NUM_POMPE_COMANDATE *)
  [ %MW1 := %MW1 - 1 ]    (* NUM_POMPE_COMANDATE, NUM_POMPE_COMANDATE *)
  // as ST:
  //   IF FALLING(P6_COMANDATA) AND NUM_POMPE_COMANDATE > 0 THEN NUM_POMPE_COMANDATE := NUM_POMPE_COMANDATE - 1; END_IF;

Subroutine Usabilità Pompe
  (* SectionNumber=10, Number=8 *)

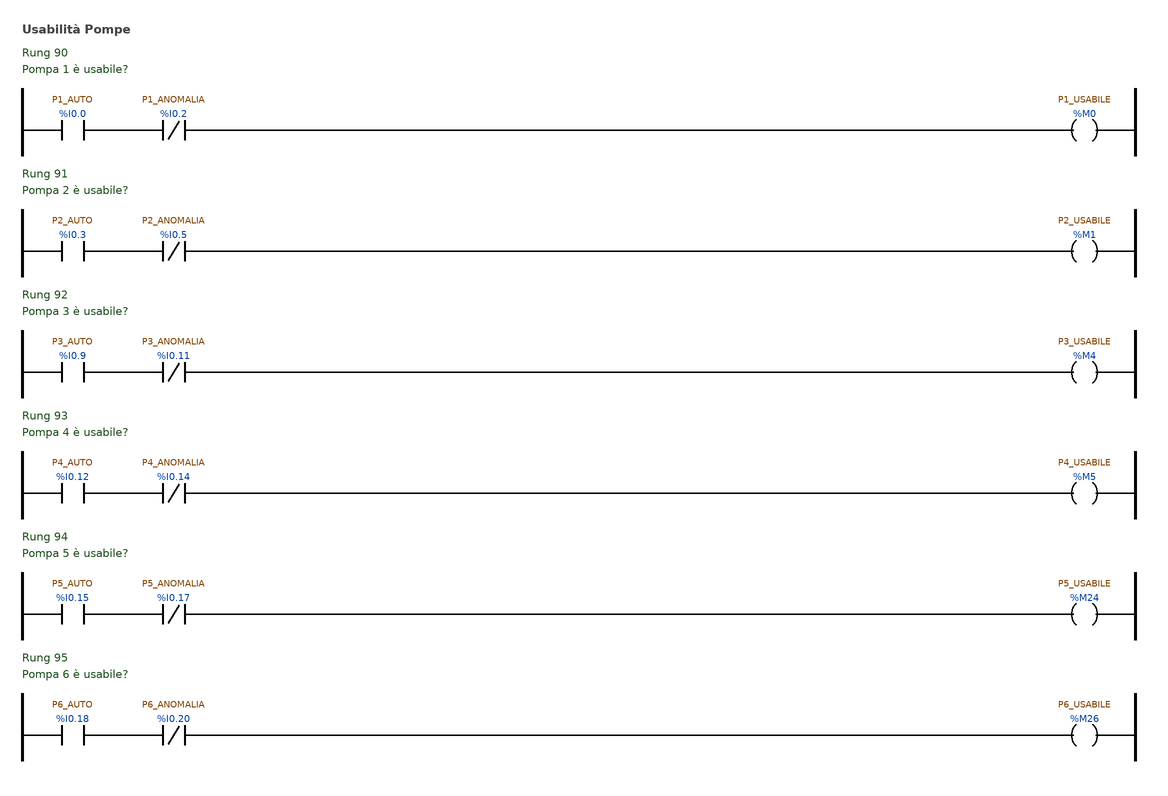

// Rung 90
// Pompa 1 è usabile?
  LD %I0.0                (* P1_AUTO *)
  ANDN %I0.2              (* P1_ANOMALIA *)
  ST %M0                  (* P1_USABILE *)
  // as ST:
  //   P1_USABILE := P1_AUTO AND NOT P1_ANOMALIA;

// Rung 91
// Pompa 2 è usabile?
  LD %I0.3                (* P2_AUTO *)
  ANDN %I0.5              (* P2_ANOMALIA *)
  ST %M1                  (* P2_USABILE *)
  // as ST:
  //   P2_USABILE := P2_AUTO AND NOT P2_ANOMALIA;

// Rung 92
// Pompa 3 è usabile?
  LD %I0.9                (* P3_AUTO *)
  ANDN %I0.11             (* P3_ANOMALIA *)
  ST %M4                  (* P3_USABILE *)
  // as ST:
  //   P3_USABILE := P3_AUTO AND NOT P3_ANOMALIA;

// Rung 93
// Pompa 4 è usabile?
  LD %I0.12               (* P4_AUTO *)
  ANDN %I0.14             (* P4_ANOMALIA *)
  ST %M5                  (* P4_USABILE *)
  // as ST:
  //   P4_USABILE := P4_AUTO AND NOT P4_ANOMALIA;

// Rung 94
// Pompa 5 è usabile?
  LD %I0.15               (* P5_AUTO *)
  ANDN %I0.17             (* P5_ANOMALIA *)
  ST %M24                 (* P5_USABILE *)
  // as ST:
  //   P5_USABILE := P5_AUTO AND NOT P5_ANOMALIA;

// Rung 95
// Pompa 6 è usabile?
  LD %I0.18               (* P6_AUTO *)
  ANDN %I0.20             (* P6_ANOMALIA *)
  ST %M26                 (* P6_USABILE *)
  // as ST:
  //   P6_USABILE := P6_AUTO AND NOT P6_ANOMALIA;

Subroutine Aggiorna Strategia Alternanza
  (* SectionNumber=11, Number=13 *)

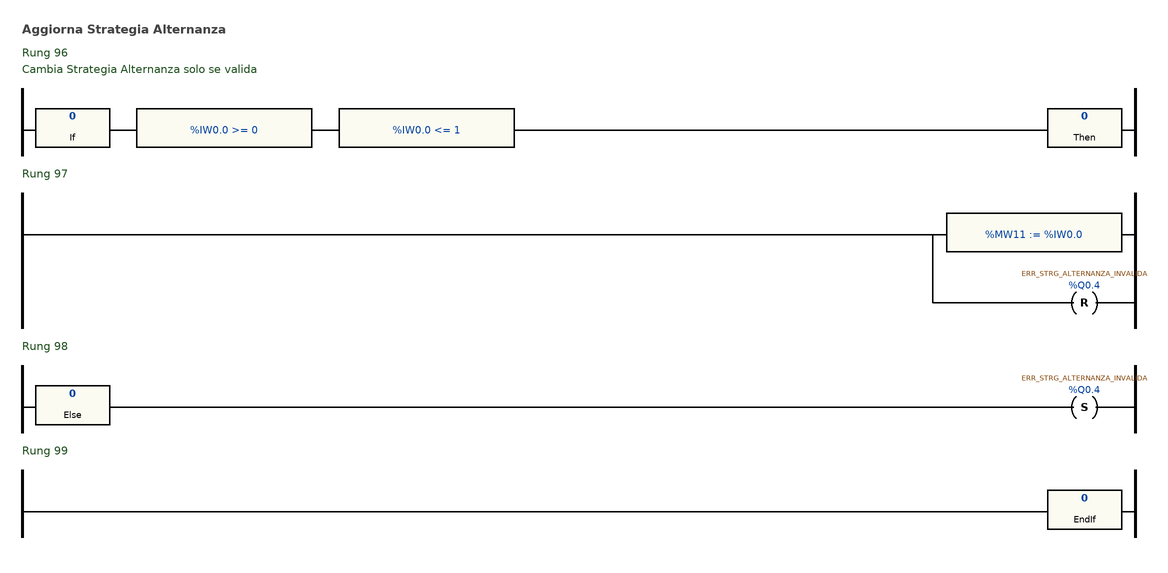

// Rung 96
// Cambia Strategia Alternanza solo se valida
  IF0
  AND [ %IW0.0 >= 0 ]     (* IO_STRG_ALTERNANZA *)
  AND [ %IW0.0 <= 1 ]     (* IO_STRG_ALTERNANZA *)
  THEN0

// Rung 97
  LD 1
  [ %MW11 := %IW0.0 ]     (* STRG_ALTERNANZA_ATTUALE, IO_STRG_ALTERNANZA *)
  R %Q0.4                 (* ERR_STRG_ALTERNANZA_INVALIDA *)
  // as ST:
  //   STRG_ALTERNANZA_ATTUALE := IO_STRG_ALTERNANZA;
  //   ERR_STRG_ALTERNANZA_INVALIDA := FALSE;

// Rung 98
  ELSE0
  S %Q0.4                 (* ERR_STRG_ALTERNANZA_INVALIDA *)

// Rung 99
  LD 1
  ENDIF0

Subroutine Soglie
  (* SectionNumber=12, Number=19 *)

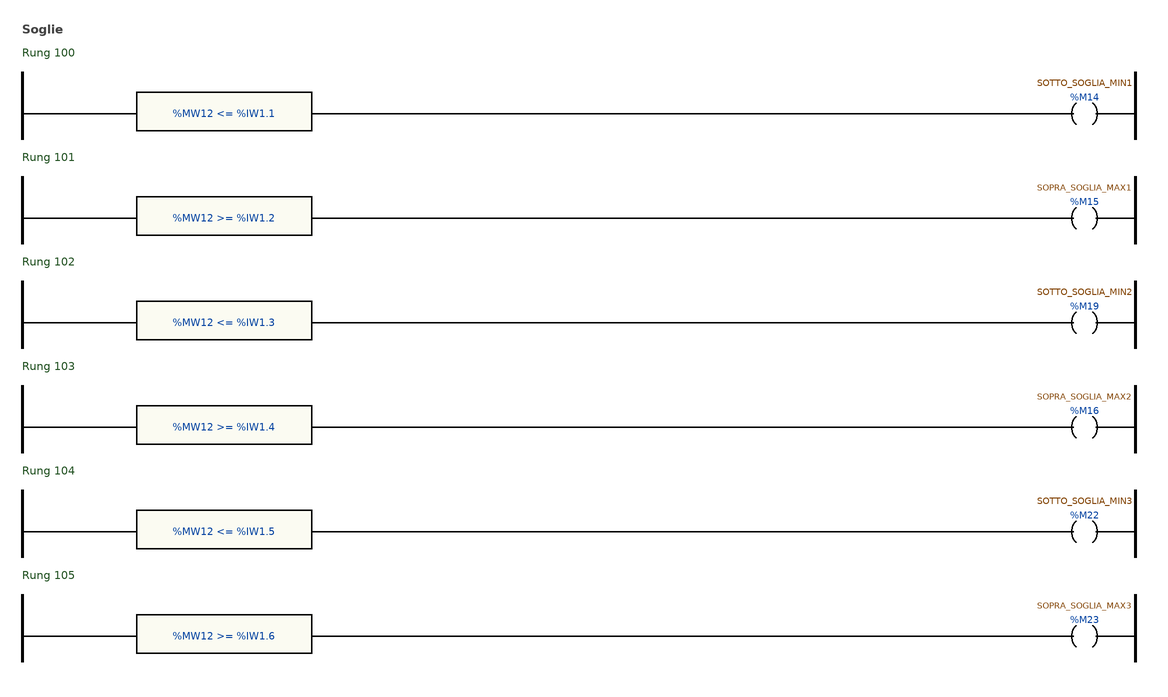

// Rung 100
  LD [ %MW12 <= %IW1.1 ]  (* LVL_PERC, SOGLIA_MIN1_PERC *)
  ST %M14                 (* SOTTO_SOGLIA_MIN1 *)
  // as ST:
  //   SOTTO_SOGLIA_MIN1 := LVL_PERC <= SOGLIA_MIN1_PERC;

// Rung 101
  LD [ %MW12 >= %IW1.2 ]  (* LVL_PERC, SOGLIA_MAX1_PERC *)
  ST %M15                 (* SOPRA_SOGLIA_MAX1 *)
  // as ST:
  //   SOPRA_SOGLIA_MAX1 := LVL_PERC >= SOGLIA_MAX1_PERC;

// Rung 102
  LD [ %MW12 <= %IW1.3 ]  (* LVL_PERC, SOGLIA_MIN2_PERC *)
  ST %M19                 (* SOTTO_SOGLIA_MIN2 *)
  // as ST:
  //   SOTTO_SOGLIA_MIN2 := LVL_PERC <= SOGLIA_MIN2_PERC;

// Rung 103
  LD [ %MW12 >= %IW1.4 ]  (* LVL_PERC, SOGLIA_MAX2_PERC *)
  ST %M16                 (* SOPRA_SOGLIA_MAX2 *)
  // as ST:
  //   SOPRA_SOGLIA_MAX2 := LVL_PERC >= SOGLIA_MAX2_PERC;

// Rung 104
  LD [ %MW12 <= %IW1.5 ]  (* LVL_PERC, SOGLIA_MIN3_PERC *)
  ST %M22                 (* SOTTO_SOGLIA_MIN3 *)
  // as ST:
  //   SOTTO_SOGLIA_MIN3 := LVL_PERC <= SOGLIA_MIN3_PERC;

// Rung 105
  LD [ %MW12 >= %IW1.6 ]  (* LVL_PERC, SOGLIA_MAX3_PERC *)
  ST %M23                 (* SOPRA_SOGLIA_MAX3 *)
  // as ST:
  //   SOPRA_SOGLIA_MAX3 := LVL_PERC >= SOGLIA_MAX3_PERC;

Subroutine Scaling
  (* SectionNumber=13, Number=20 *)

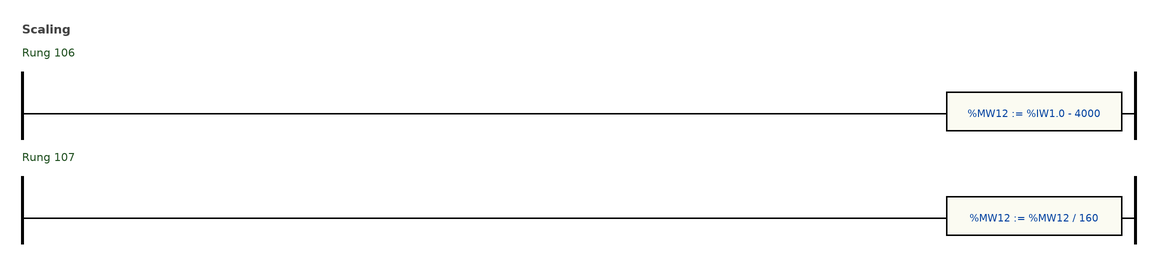

// Rung 106
  LD 1
  [ %MW12 := %IW1.0 - 4000 ](* LVL_PERC, IO_LVL *)
  // as ST:
  //   LVL_PERC := IO_LVL - 4000;

// Rung 107
  LD 1
  [ %MW12 := %MW12 / 160 ](* LVL_PERC, LVL_PERC *)
  // as ST:
  //   LVL_PERC := LVL_PERC / 160;

Subroutine Quante Pompe da Comandare (Livello minimo)
  (* SectionNumber=14, Number=9 *)

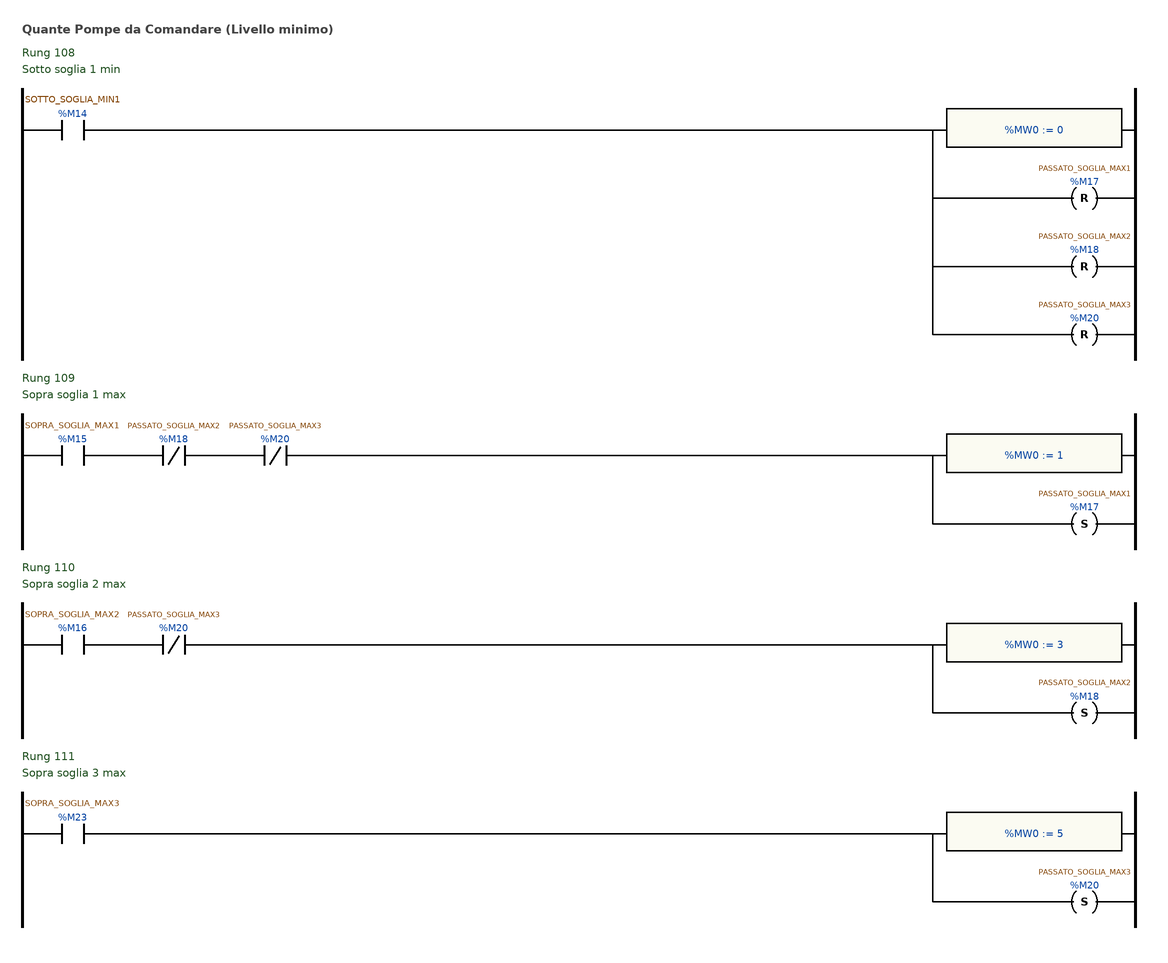

// Rung 108
// Sotto soglia 1 min
  LD %M14                 (* SOTTO_SOGLIA_MIN1 *)
  [ %MW0 := 0 ]           (* NUM_POMPE_DA_COMANDARE *)
  R %M17                  (* PASSATO_SOGLIA_MAX1 *)
  R %M18                  (* PASSATO_SOGLIA_MAX2 *)
  R %M20                  (* PASSATO_SOGLIA_MAX3 *)
  // as ST:
  //   IF SOTTO_SOGLIA_MIN1 THEN NUM_POMPE_DA_COMANDARE := 0; END_IF;
  //   IF SOTTO_SOGLIA_MIN1 THEN PASSATO_SOGLIA_MAX1 := FALSE; END_IF;
  //   IF SOTTO_SOGLIA_MIN1 THEN PASSATO_SOGLIA_MAX2 := FALSE; END_IF;
  //   IF SOTTO_SOGLIA_MIN1 THEN PASSATO_SOGLIA_MAX3 := FALSE; END_IF;

// Rung 109
// Sopra soglia 1 max
  LD %M15                 (* SOPRA_SOGLIA_MAX1 *)
  ANDN %M18               (* PASSATO_SOGLIA_MAX2 *)
  ANDN %M20               (* PASSATO_SOGLIA_MAX3 *)
  [ %MW0 := 1 ]           (* NUM_POMPE_DA_COMANDARE *)
  S %M17                  (* PASSATO_SOGLIA_MAX1 *)
  // as ST:
  //   IF SOPRA_SOGLIA_MAX1 AND NOT PASSATO_SOGLIA_MAX2 AND NOT PASSATO_SOGLIA_MAX3 THEN NUM_POMPE_DA_COMANDARE := 1; END_IF;
  //   IF SOPRA_SOGLIA_MAX1 AND NOT PASSATO_SOGLIA_MAX2 AND NOT PASSATO_SOGLIA_MAX3 THEN PASSATO_SOGLIA_MAX1 := TRUE; END_IF;

// Rung 110
// Sopra soglia 2 max
  LD %M16                 (* SOPRA_SOGLIA_MAX2 *)
  ANDN %M20               (* PASSATO_SOGLIA_MAX3 *)
  [ %MW0 := 3 ]           (* NUM_POMPE_DA_COMANDARE *)
  S %M18                  (* PASSATO_SOGLIA_MAX2 *)
  // as ST:
  //   IF SOPRA_SOGLIA_MAX2 AND NOT PASSATO_SOGLIA_MAX3 THEN NUM_POMPE_DA_COMANDARE := 3; END_IF;
  //   IF SOPRA_SOGLIA_MAX2 AND NOT PASSATO_SOGLIA_MAX3 THEN PASSATO_SOGLIA_MAX2 := TRUE; END_IF;

// Rung 111
// Sopra soglia 3 max
  LD %M23                 (* SOPRA_SOGLIA_MAX3 *)
  [ %MW0 := 5 ]           (* NUM_POMPE_DA_COMANDARE *)
  S %M20                  (* PASSATO_SOGLIA_MAX3 *)
  // as ST:
  //   IF SOPRA_SOGLIA_MAX3 THEN NUM_POMPE_DA_COMANDARE := 5; END_IF;
  //   IF SOPRA_SOGLIA_MAX3 THEN PASSATO_SOGLIA_MAX3 := TRUE; END_IF;

Subroutine Quante Pompe da Comandare (Spegnimento graduale)
  (* SectionNumber=15, Number=10 *)

